// TIA Portal project "PP_0.25AC_new" (V14)

(* hardware
DEVICE "S7-1200 station_1"  S7-1200 Station
   slot 0: "Rack_0"  Rack  V1.0
   slot 1: "PLC_1"  CPU 1215C DC/DC/DC  6ES7 215-1AG40-0XB0  V4.2
   slot 101: "CM 1241 (RS422/485)_1"  6ES7 241-1CH31-0XB0  V1.0
DEVICE "ET 200SP station_1"  ET 200SP-Station
   slot 0: "Rack_0"  Rack  6ES5 710-8MAx1
   slot 0: "IO device_1"  IM 155-6 PN ST  6ES7 155-6AU01-0BN0  V4.1
   slot 1: "AI 8xI 2-,4-wire BA_1"  AI 8xI 2-,4-wire BA  6ES7 134-6GF00-0AA1  V1.0
      slot 1: "AI 8xI 2-,4-wire BA_1"  AI 8xI 2-,4-wire BA
   slot 2: "AI 8xI 2-,4-wire BA_2"  AI 8xI 2-,4-wire BA  6ES7 134-6GF00-0AA1  V1.0
      slot 1: "AI 8xI 2-,4-wire BA_2"  AI 8xI 2-,4-wire BA
   slot 3: "Server module_1"  Server module  6ES7 193-6PA00-0AA0  V1.1
      slot 1: "Server module_1"  Server module
   slot 127: "BA 2xRJ45"  BA 2xRJ45  6ES7 193-6AR00-0AA0  V0.0
      slot 1: "Port_1"  6ES7 193-6AR00-0AA0  V0.0
      slot 2: "Port_2"  6ES7 193-6AR00-0AA0  V0.0
*)

// ===== PLC "PLC_1"  CPU 1215C DC/DC/DC =====

VAR_GLOBAL   // PLC tag table "Default tag table"
   "AI2_0" AT %IW2 : Int;   // Давление нефти на входе, МПа
   "AI2_1" AT %IW4 : Int;   // Давление нефти на выходе, МПа
   "AI2_2" AT %IW6 : Int;   // Давление газа, МПа
   "AI2_3" AT %IW8 : Int;   // Температура на выходе, С
   "AI2_4" AT %IW10 : Int;   // Температура дымовых газов горелки, С
   "AI2_5" AT %IW12 : Int;   // Температура ёмкости, С
   "AI2_6" AT %IW14 : Int;   // Температура в емкости Б1, С ТТ3
   "AI2_7" AT %IW16 : Int;   // Газоанализатор
   "AI3_0" AT %IW18 : Int;   // Резерв
   "AI3_1" AT %IW20 : Int;   // Резерв
   "AI3_2" AT %IW22 : Int;   // Резерв
   "AI3_3" AT %IW24 : Int;   // Резерв
   "AI3_4" AT %IW26 : Int;   // Резерв
   "AI3_5" AT %IW28 : Int;   // Резерв
   "AI3_6" AT %IW30 : Int;   // Резерв
   "AI3_7" AT %IW32 : Int;   // Резерв
   "DI1_0" AT %I0.0 : Bool;   // Сигнализатор уровня MIN ёмкости
   "DI1_1" AT %I0.1 : Bool;   // Сигнализатор уровня MAX ёмкости
   "DI1_2" AT %I0.2 : Bool;   // Клапан 1
   "DI1_3" AT %I0.3 : Bool;   // Клапан 2
   "DI1_4" AT %I0.4 : Bool;   // Резерв
   "DI1_5" AT %I0.5 : Bool;   // Резерв
   "DI1_6" AT %I0.6 : Bool;   // Работа горелки
   "DI1_7" AT %I0.7 : Bool;   // Авария горелки
   "DI1_8" AT %I1.0 : Bool;   // Резерв
   "DI1_9" AT %I1.1 : Bool;   // Резерв
   "DI1_10" AT %I1.2 : Bool;   // Резерв
   "DI1_11" AT %I1.3 : Bool;   // Резерв
   "DI1_12" AT %I1.4 : Bool;   // Резерв
   "DI1_13" AT %I1.5 : Bool;   // Резерв
   "DI2_0" AT %I48.0 : Bool;   // Резерв
   "DI2_1" AT %I48.1 : Bool;   // Резерв
   "DI2_2" AT %I48.2 : Bool;   // Резерв
   "DI2_3" AT %I48.3 : Bool;   // Резерв
   "DI2_4" AT %I48.4 : Bool;   // Резерв
   "DI2_5" AT %I48.5 : Bool;   // Резерв
   "DI2_6" AT %I48.6 : Bool;   // Резерв
   "DI2_7" AT %I48.7 : Bool;   // Резерв
   "DI2_8" AT %I49.0 : Bool;   // Резерв
   "DI2_9" AT %I49.1 : Bool;   // Резерв
   "DI2_10" AT %I49.2 : Bool;   // Резерв
   "DI2_11" AT %I49.3 : Bool;   // Резерв
   "DI2_12" AT %I49.4 : Bool;   // Резерв
   "DI2_13" AT %I49.5 : Bool;   // Резерв
   "DI2_14" AT %I49.6 : Bool;   // Резерв
   "DI2_15" AT %I49.7 : Bool;   // Резерв
   "DO1_0" AT %Q0.0 : Bool;   // ПАСВ оповещатель светозвуковой
   "DO1_1" AT %Q0.1 : Bool;   // ПАСВ оповещатель светозвуковой
   "DO1_2" AT %Q0.2 : Bool;   // Пуск/Стоп горелки
   "DO1_3" AT %Q0.3 : Bool;   // Клапан 1
   "DO1_4" AT %Q0.4 : Bool;   // Клапан 2
   "DO1_5" AT %Q0.5 : Bool;   // ИВНТР
   "DO1_6" AT %Q0.6 : Bool;   // Резерв
   "DO1_7" AT %Q0.7 : Bool;   // Резерв
   "DO1_8" AT %Q1.0 : Bool;   // Резерв
   "DO1_9" AT %Q1.1 : Bool;   // Резерв
   "DO2_0" AT %Q2.0 : Bool;   // Резерв
   "DO2_1" AT %Q2.1 : Bool;   // Резерв
   "DO2_2" AT %Q2.2 : Bool;   // Резерв
   "DO2_3" AT %Q2.3 : Bool;   // Резерв
   "DO2_4" AT %Q2.4 : Bool;   // Резерв
   "DO2_5" AT %Q2.5 : Bool;   // Резерв
   "DO2_6" AT %Q2.6 : Bool;   // Резерв
   "DO2_7" AT %Q2.7 : Bool;   // Резерв
   "DO2_8" AT %Q3.0 : Bool;   // Резерв
   "DO2_9" AT %Q3.1 : Bool;   // Резерв
   "DO2_10" AT %Q3.2 : Bool;   // Резерв
   "DO2_11" AT %Q3.3 : Bool;   // Резерв
   "DO2_12" AT %Q3.4 : Bool;   // Резерв
   "DO2_13" AT %Q3.5 : Bool;   // Резерв
   "DO2_14" AT %Q3.6 : Bool;   // Резерв
   "DO2_15" AT %Q3.7 : Bool;   // Резерв
   "Clock_Byte" AT %MB0 : Byte;
   "Clock_10Hz" AT %M0.0 : Bool;
   "Clock_5Hz" AT %M0.1 : Bool;
   "Clock_2.5Hz" AT %M0.2 : Bool;
   "Clock_2Hz" AT %M0.3 : Bool;
   "Clock_1.25Hz" AT %M0.4 : Bool;
   "Clock_1Hz" AT %M0.5 : Bool;
   "Clock_0.625Hz" AT %M0.6 : Bool;
   "Clock_0.5Hz" AT %M0.7 : Bool;
   "System_Byte" AT %MB1 : Byte;
   "FirstScan" AT %M1.0 : Bool;
   "DiagStatusUpdate" AT %M1.1 : Bool;
   "AlwaysTRUE" AT %M1.2 : Bool;
   "AlwaysFALSE" AT %M1.3 : Bool;
   "EN" AT %M2.0 : Bool;
END_VAR

TYPE "Burner_DT"
VERSION : 0.1
   STRUCT
      State : Int;
      CMD_in : Int;
      Alarm : Int;
   END_STRUCT;
END_TYPE

TYPE "AI_DT"
VERSION : 0.1
   STRUCT
      Hihi_Value : Real;   // Уставка: Hihi
      High_Value : Real;   // Уставка: High
      Low_Value : Real;   // Уставка: Low
      Lolo_Value : Real;   // Уставка: Lolo
      MIN_Current : Real;   // Настройка: Минимальное входное значение тока
      MAX_Current : Real;   // Настройка: Максимальное входное значение тока
      MAX_Value : Real;   // Настройка: Максимальное значение измеряемой величины
      MIN_Value : Real;   // Настройка: Минимальное значение измеряемой величины
      Underflow_RAW : Real;   // Настройка: Значение кода ацп при обрыве
      Overflow_RAW : Real;   // Настройка: Значение кода ацп при зашкале
      SCALED : Real;   // Выход: Масштабированное в инженерные единицы значение входного сигнала
      ING_Value : Real;   // Выход: Токовое значение датчика
      Manual_Value : Real;   // Значение, введенное вручную
      Alarm_Delay : Int;   // Настройка: Задержка срабатывания аварий
      Warning_Delay : Int;   // Настройка: Задержка срабатывания предупреждений
      AVG_Delay : Real;   // Настройка: Зона нечувствительности
      Underflow_Delay : Int;   // Настройка: Задержка отображения обрыва датчика
      Overflow_Delay : Int;   // Настройка: Задержка отображения неисправности датчика
      State : Word;   // Выход: Состояние датчика
      Modeee : Word;   // Настройка: Режим работы датчика
      bools : Word;   // Все булевы параметры AI
      AI_RAW_MIN : Int;   // Мин кода ацп
      AI_RAW_MAX : Int;   // Макс кода ацп
      Hihi_EN : Bool;   // Разрешение на сработку
      High_EN : Bool;   // Разрешение на сработку
      Low_En : Bool;   // Разрешение на сработку
      Lolo_EN : Bool;   // Разрешение на сработку
   END_STRUCT;
END_TYPE

TYPE "Ustavki"
   STRUCT
      Hihi : Bool;
      Hi : Bool;
      Lo : Bool;
      Lolo : Bool;
   END_STRUCT;
END_TYPE

TYPE "PAZ_DT"
VERSION : 0.1
   STRUCT
      Alarm_EN : Bool;
      ZP_EN : Bool;
      IN : Bool;
      Alarm_out : Bool;
      ZP_out : Bool;
   END_STRUCT;
END_TYPE

TYPE "Hiter"
VERSION : 0.1
   STRUCT
      Mode : Bool;
      T_state : Int;
      CMD : Bool;
      Avar_stop : Bool;
   END_STRUCT;
END_TYPE

TYPE "DI_DT"
VERSION : 0.1
   STRUCT
      Time_ON : Int;   // Время перехода OFF->ON
      Time_OFF : Int;   // Время перехода ON->OFF
      Input : Bool;   // Значение с модуля
      Disable : Bool;   // Запрет обработки канала
      Invert : Bool;   // Инертирование канала
      Output : Bool;   // Значение канала для логики
   END_STRUCT;
END_TYPE

TYPE "Valve_DT"
VERSION : 0.1
   STRUCT
      State : Int;
      State_ctrl : Bool;
      Alarm : Int;
      Cmd_in : Int;
      Cmd_out : Bool;
      bools : Int;
      Deblock : Bool;
   END_STRUCT;
END_TYPE

TYPE "Valve_ctrl_DT"
VERSION : 0.1
   STRUCT
      State : Int;
      Cmd_in : Int;
      TIME_shod : Int;
      TIME_hod : Int;
      bools : DWord;
   END_STRUCT;
END_TYPE

TYPE "DO_DT"
VERSION : 0.1
   STRUCT
      Time_ON : Int;   // Время перехода OFF->ON
      Time_OFF : Int;   // Время перехода ON->OFF
      Input : Bool;   // Значение от логики
      Disable : Bool;   // Запрет обработки канала
      Invert : Bool;   // Инертирование канала
      Output : Bool;   // Значение на модуль
   END_STRUCT;
END_TYPE

DATA_BLOCK "PLC_Signals_DB"   // DB1
{ S7_Optimized_Access := 'FALSE' }
VERSION : 0.1
   VAR
      AI_2_0 : Struct   // Давление на выходе
         Hihi_Value : Real := 70.0;   // Уставка: Hihi
         High_Value : Real := 60.0;   // Уставка: High
         Low_Value : Real := 30.0;   // Уставка: Low
         Lolo_Value : Real := 20.0;   // Уставка: Lolo
         MIN_Current : Real := 4.0;   // Настройка: Минимальное входное значение тока
         MAX_Current : Real := 20.0;   // Настройка: Максимальное входное значение тока
         MAX_Value : Real := 1.0;   // Настройка: Максимальное значение измеряемой величины
         MIN_Value : Real := 0.0;   // Настройка: Минимальное значение измеряемой величины
         Underflow_RAW : Real := -10.0;   // Настройка: Значение кода ацп при обрыве
         Overflow_RAW : Real := 27650.0;   // Настройка: Значение кода ацп при зашкале
         SCALED : Real := 0.0;   // Выход: Масштабированное в инженерные единицы значение входного сигнала
         ING_Value : Real := 0.0;   // Выход: Токовое значение датчика
         Manual_Value : Real := 50.0;   // Значение, введенное вручную
         Alarm_Delay : Int := 0;   // Настройка: Задержка срабатывания аварий
         Warning_Delay : Int := 0;   // Настройка: Задержка срабатывания предупреждений
         AVG_Delay : Real := 0.0;   // Настройка: Зона нечувствительности
         Underflow_Delay : Int := 0;   // Настройка: Задержка отображения обрыва датчика
         Overflow_Delay : Int := 0;   // Настройка: Задержка отображения неисправности датчика
         StateHMI : Int;
         State : Word := 16#0;   // Выход: Состояние датчика
         Modeee : Word := 16#1;   // Настройка: Режим работы датчика
         bools : Word := 16#0;   // Все булевы параметры AI
         AI_RAW_MIN : Int := 0;   // Мин кода ацп
         AI_RAW_MAX : Int := 27648;   // Макс кода ацп
         Hihi_EN : Bool := false;   // Разрешение на сработку
         High_EN : Bool := false;   // Разрешение на сработку
         Low_En : Bool := false;   // Разрешение на сработку
         Lolo_EN : Bool := false;   // Разрешение на сработку
      END_STRUCT;
      AI_2_1 : Struct   // Давление на входе
         Hihi_Value : Real := 70.0;   // Уставка: Hihi
         High_Value : Real := 60.0;   // Уставка: High
         Low_Value : Real := 30.0;   // Уставка: Low
         Lolo_Value : Real := 20.0;   // Уставка: Lolo
         MIN_Current : Real := 4.0;   // Настройка: Минимальное входное значение тока
         MAX_Current : Real := 20.0;   // Настройка: Максимальное входное значение тока
         MAX_Value : Real := 1.0;   // Настройка: Максимальное значение измеряемой величины
         MIN_Value : Real := 0.0;   // Настройка: Минимальное значение измеряемой величины
         Underflow_RAW : Real := -10.0;   // Настройка: Значение кода ацп при обрыве
         Overflow_RAW : Real := 27650.0;   // Настройка: Значение кода ацп при зашкале
         SCALED : Real := 0.0;   // Выход: Масштабированное в инженерные единицы значение входного сигнала
         ING_Value : Real := 0.0;   // Выход: Токовое значение датчика
         Manual_Value : Real := 50.0;   // Значение, введенное вручную
         Alarm_Delay : Int := 0;   // Настройка: Задержка срабатывания аварий
         Warning_Delay : Int := 0;   // Настройка: Задержка срабатывания предупреждений
         AVG_Delay : Real := 0.0;   // Настройка: Зона нечувствительности
         Underflow_Delay : Int := 0;   // Настройка: Задержка отображения обрыва датчика
         Overflow_Delay : Int := 0;   // Настройка: Задержка отображения неисправности датчика
         StateHMI : Int;
         State : Word := 16#0;   // Выход: Состояние датчика
         Modeee : Word := 16#1;   // Настройка: Режим работы датчика
         bools : Word := 16#0;   // Все булевы параметры AI
         AI_RAW_MIN : Int := 0;   // Мин кода ацп
         AI_RAW_MAX : Int := 27648;   // Макс кода ацп
         Hihi_EN : Bool := false;   // Разрешение на сработку
         High_EN : Bool := false;   // Разрешение на сработку
         Low_En : Bool := false;   // Разрешение на сработку
         Lolo_EN : Bool := false;   // Разрешение на сработку
      END_STRUCT;
      AI_2_2 : Struct   // Датчик давления газа
         Hihi_Value : Real := 70.0;   // Уставка: Hihi
         High_Value : Real := 60.0;   // Уставка: High
         Low_Value : Real := 30.0;   // Уставка: Low
         Lolo_Value : Real := 20.0;   // Уставка: Lolo
         MIN_Current : Real := 4.0;   // Настройка: Минимальное входное значение тока
         MAX_Current : Real := 20.0;   // Настройка: Максимальное входное значение тока
         MAX_Value : Real := 1.0;   // Настройка: Максимальное значение измеряемой величины
         MIN_Value : Real := 0.0;   // Настройка: Минимальное значение измеряемой величины
         Underflow_RAW : Real := -10.0;   // Настройка: Значение кода ацп при обрыве
         Overflow_RAW : Real := 27650.0;   // Настройка: Значение кода ацп при зашкале
         SCALED : Real := 0.0;   // Выход: Масштабированное в инженерные единицы значение входного сигнала
         ING_Value : Real := 0.0;   // Выход: Токовое значение датчика
         Manual_Value : Real := 50.0;   // Значение, введенное вручную
         Alarm_Delay : Int := 0;   // Настройка: Задержка срабатывания аварий
         Warning_Delay : Int := 0;   // Настройка: Задержка срабатывания предупреждений
         AVG_Delay : Real := 0.0;   // Настройка: Зона нечувствительности
         Underflow_Delay : Int := 0;   // Настройка: Задержка отображения обрыва датчика
         Overflow_Delay : Int := 0;   // Настройка: Задержка отображения неисправности датчика
         StateHMI : Int;
         State : Word := 16#0;   // Выход: Состояние датчика
         Modeee : Word := 16#1;   // Настройка: Режим работы датчика
         bools : Word := 16#0;   // Все булевы параметры AI
         AI_RAW_MIN : Int := 0;   // Мин кода ацп
         AI_RAW_MAX : Int := 27648;   // Макс кода ацп
         Hihi_EN : Bool := false;   // Разрешение на сработку
         High_EN : Bool := false;   // Разрешение на сработку
         Low_En : Bool := false;   // Разрешение на сработку
         Lolo_EN : Bool := false;   // Разрешение на сработку
      END_STRUCT;
      AI_2_3 : Struct   // Температура на выходе
         Hihi_Value : Real := 70.0;   // Уставка: Hihi
         High_Value : Real := 60.0;   // Уставка: High
         Low_Value : Real := 30.0;   // Уставка: Low
         Lolo_Value : Real := 20.0;   // Уставка: Lolo
         MIN_Current : Real := 4.0;   // Настройка: Минимальное входное значение тока
         MAX_Current : Real := 20.0;   // Настройка: Максимальное входное значение тока
         MAX_Value : Real := 100.0;   // Настройка: Максимальное значение измеряемой величины
         MIN_Value : Real := -50.0;   // Настройка: Минимальное значение измеряемой величины
         Underflow_RAW : Real := -10.0;   // Настройка: Значение кода ацп при обрыве
         Overflow_RAW : Real := 27650.0;   // Настройка: Значение кода ацп при зашкале
         SCALED : Real := 0.0;   // Выход: Масштабированное в инженерные единицы значение входного сигнала
         ING_Value : Real := 0.0;   // Выход: Токовое значение датчика
         Manual_Value : Real := 50.0;   // Значение, введенное вручную
         Alarm_Delay : Int := 0;   // Настройка: Задержка срабатывания аварий
         Warning_Delay : Int := 0;   // Настройка: Задержка срабатывания предупреждений
         AVG_Delay : Real := 0.0;   // Настройка: Зона нечувствительности
         Underflow_Delay : Int := 0;   // Настройка: Задержка отображения обрыва датчика
         Overflow_Delay : Int := 0;   // Настройка: Задержка отображения неисправности датчика
         StateHMI : Int;
         State : Word := 16#0;   // Выход: Состояние датчика
         Modeee : Word := 16#1;   // Настройка: Режим работы датчика
         bools : Word := 16#0;   // Все булевы параметры AI
         AI_RAW_MIN : Int := 0;   // Мин кода ацп
         AI_RAW_MAX : Int := 27648;   // Макс кода ацп
         Hihi_EN : Bool := false;   // Разрешение на сработку
         High_EN : Bool := false;   // Разрешение на сработку
         Low_En : Bool := false;   // Разрешение на сработку
         Lolo_EN : Bool := false;   // Разрешение на сработку
      END_STRUCT;
      AI_2_4 : Struct   // Температура дымовых газов
         Hihi_Value : Real := 70.0;   // Уставка: Hihi
         High_Value : Real := 60.0;   // Уставка: High
         Low_Value : Real := 30.0;   // Уставка: Low
         Lolo_Value : Real := 20.0;   // Уставка: Lolo
         MIN_Current : Real := 4.0;   // Настройка: Минимальное входное значение тока
         MAX_Current : Real := 20.0;   // Настройка: Максимальное входное значение тока
         MAX_Value : Real := 500.0;   // Настройка: Максимальное значение измеряемой величины
         MIN_Value : Real := -50.0;   // Настройка: Минимальное значение измеряемой величины
         Underflow_RAW : Real := -10.0;   // Настройка: Значение кода ацп при обрыве
         Overflow_RAW : Real := 27650.0;   // Настройка: Значение кода ацп при зашкале
         SCALED : Real := 0.0;   // Выход: Масштабированное в инженерные единицы значение входного сигнала
         ING_Value : Real := 0.0;   // Выход: Токовое значение датчика
         Manual_Value : Real := 50.0;   // Значение, введенное вручную
         Alarm_Delay : Int := 0;   // Настройка: Задержка срабатывания аварий
         Warning_Delay : Int := 0;   // Настройка: Задержка срабатывания предупреждений
         AVG_Delay : Real := 0.0;   // Настройка: Зона нечувствительности
         Underflow_Delay : Int := 0;   // Настройка: Задержка отображения обрыва датчика
         Overflow_Delay : Int := 0;   // Настройка: Задержка отображения неисправности датчика
         StateHMI : Int;
         State : Word := 16#0;   // Выход: Состояние датчика
         Modeee : Word := 16#1;   // Настройка: Режим работы датчика
         bools : Word := 16#0;   // Все булевы параметры AI
         AI_RAW_MIN : Int := 0;   // Мин кода ацп
         AI_RAW_MAX : Int := 27648;   // Макс кода ацп
         Hihi_EN : Bool := false;   // Разрешение на сработку
         High_EN : Bool := false;   // Разрешение на сработку
         Low_En : Bool := false;   // Разрешение на сработку
         Lolo_EN : Bool := false;   // Разрешение на сработку
      END_STRUCT;
      AI_2_5 : Struct   // Температура ёмкости
         Hihi_Value : Real := 70.0;   // Уставка: Hihi
         High_Value : Real := 60.0;   // Уставка: High
         Low_Value : Real := 30.0;   // Уставка: Low
         Lolo_Value : Real := 20.0;   // Уставка: Lolo
         MIN_Current : Real := 4.0;   // Настройка: Минимальное входное значение тока
         MAX_Current : Real := 20.0;   // Настройка: Максимальное входное значение тока
         MAX_Value : Real := 100.0;   // Настройка: Максимальное значение измеряемой величины
         MIN_Value : Real := -50.0;   // Настройка: Минимальное значение измеряемой величины
         Underflow_RAW : Real := -10.0;   // Настройка: Значение кода ацп при обрыве
         Overflow_RAW : Real := 27650.0;   // Настройка: Значение кода ацп при зашкале
         SCALED : Real := 0.0;   // Выход: Масштабированное в инженерные единицы значение входного сигнала
         ING_Value : Real := 0.0;   // Выход: Токовое значение датчика
         Manual_Value : Real := 50.0;   // Значение, введенное вручную
         Alarm_Delay : Int := 0;   // Настройка: Задержка срабатывания аварий
         Warning_Delay : Int := 0;   // Настройка: Задержка срабатывания предупреждений
         AVG_Delay : Real := 0.0;   // Настройка: Зона нечувствительности
         Underflow_Delay : Int := 0;   // Настройка: Задержка отображения обрыва датчика
         Overflow_Delay : Int := 0;   // Настройка: Задержка отображения неисправности датчика
         StateHMI : Int;
         State : Word := 16#0;   // Выход: Состояние датчика
         Modeee : Word := 16#1;   // Настройка: Режим работы датчика
         bools : Word := 16#0;   // Все булевы параметры AI
         AI_RAW_MIN : Int := 0;   // Мин кода ацп
         AI_RAW_MAX : Int := 27648;   // Макс кода ацп
         Hihi_EN : Bool := false;   // Разрешение на сработку
         High_EN : Bool := false;   // Разрешение на сработку
         Low_En : Bool := false;   // Разрешение на сработку
         Lolo_EN : Bool := false;   // Разрешение на сработку
      END_STRUCT;
      AI_2_6 : Struct   // Газоанализатор ДГС
         Hihi_Value : Real := 70.0;   // Уставка: Hihi
         High_Value : Real := 60.0;   // Уставка: High
         Low_Value : Real := 30.0;   // Уставка: Low
         Lolo_Value : Real := 20.0;   // Уставка: Lolo
         MIN_Current : Real := 4.0;   // Настройка: Минимальное входное значение тока
         MAX_Current : Real := 20.0;   // Настройка: Максимальное входное значение тока
         MAX_Value : Real := 100.0;   // Настройка: Максимальное значение измеряемой величины
         MIN_Value : Real := -50.0;   // Настройка: Минимальное значение измеряемой величины
         Underflow_RAW : Real := -10.0;   // Настройка: Значение кода ацп при обрыве
         Overflow_RAW : Real := 27650.0;   // Настройка: Значение кода ацп при зашкале
         SCALED : Real := 0.0;   // Выход: Масштабированное в инженерные единицы значение входного сигнала
         ING_Value : Real := 0.0;   // Выход: Токовое значение датчика
         Manual_Value : Real := 50.0;   // Значение, введенное вручную
         Alarm_Delay : Int := 0;   // Настройка: Задержка срабатывания аварий
         Warning_Delay : Int := 0;   // Настройка: Задержка срабатывания предупреждений
         AVG_Delay : Real := 0.0;   // Настройка: Зона нечувствительности
         Underflow_Delay : Int := 0;   // Настройка: Задержка отображения обрыва датчика
         Overflow_Delay : Int := 0;   // Настройка: Задержка отображения неисправности датчика
         StateHMI : Int;
         State : Word := 16#0;   // Выход: Состояние датчика
         Modeee : Word := 16#1;   // Настройка: Режим работы датчика
         bools : Word := 16#0;   // Все булевы параметры AI
         AI_RAW_MIN : Int := 0;   // Мин кода ацп
         AI_RAW_MAX : Int := 27648;   // Макс кода ацп
         Hihi_EN : Bool := false;   // Разрешение на сработку
         High_EN : Bool := false;   // Разрешение на сработку
         Low_En : Bool := false;   // Разрешение на сработку
         Lolo_EN : Bool := false;   // Разрешение на сработку
      END_STRUCT;
      AI_2_7 : Struct   // Резерв
         Hihi_Value : Real := 70.0;   // Уставка: Hihi
         High_Value : Real := 60.0;   // Уставка: High
         Low_Value : Real := 30.0;   // Уставка: Low
         Lolo_Value : Real := 20.0;   // Уставка: Lolo
         MIN_Current : Real := 4.0;   // Настройка: Минимальное входное значение тока
         MAX_Current : Real := 20.0;   // Настройка: Максимальное входное значение тока
         MAX_Value : Real := 100.0;   // Настройка: Максимальное значение измеряемой величины
         MIN_Value : Real := 0.0;   // Настройка: Минимальное значение измеряемой величины
         Underflow_RAW : Real := -10.0;   // Настройка: Значение кода ацп при обрыве
         Overflow_RAW : Real := 27650.0;   // Настройка: Значение кода ацп при зашкале
         SCALED : Real := 0.0;   // Выход: Масштабированное в инженерные единицы значение входного сигнала
         ING_Value : Real := 0.0;   // Выход: Токовое значение датчика
         Manual_Value : Real := 50.0;   // Значение, введенное вручную
         Alarm_Delay : Int := 0;   // Настройка: Задержка срабатывания аварий
         Warning_Delay : Int := 0;   // Настройка: Задержка срабатывания предупреждений
         AVG_Delay : Real := 0.0;   // Настройка: Зона нечувствительности
         Underflow_Delay : Int := 0;   // Настройка: Задержка отображения обрыва датчика
         Overflow_Delay : Int := 0;   // Настройка: Задержка отображения неисправности датчика
         StateHMI : Int;
         State : Word := 16#0;   // Выход: Состояние датчика
         Modeee : Word := 16#1;   // Настройка: Режим работы датчика
         bools : Word := 16#0;   // Все булевы параметры AI
         AI_RAW_MIN : Int := 0;   // Мин кода ацп
         AI_RAW_MAX : Int := 27648;   // Макс кода ацп
         Hihi_EN : Bool := false;   // Разрешение на сработку
         High_EN : Bool := false;   // Разрешение на сработку
         Low_En : Bool := false;   // Разрешение на сработку
         Lolo_EN : Bool := false;   // Разрешение на сработку
      END_STRUCT;
      AI_3_0 : Struct   // Резерв
         Hihi_Value : Real := 70.0;   // Уставка: Hihi
         High_Value : Real := 60.0;   // Уставка: High
         Low_Value : Real := 30.0;   // Уставка: Low
         Lolo_Value : Real := 20.0;   // Уставка: Lolo
         MIN_Current : Real := 4.0;   // Настройка: Минимальное входное значение тока
         MAX_Current : Real := 20.0;   // Настройка: Максимальное входное значение тока
         MAX_Value : Real := 100.0;   // Настройка: Максимальное значение измеряемой величины
         MIN_Value : Real := 0.0;   // Настройка: Минимальное значение измеряемой величины
         Underflow_RAW : Real := -10.0;   // Настройка: Значение кода ацп при обрыве
         Overflow_RAW : Real := 27650.0;   // Настройка: Значение кода ацп при зашкале
         SCALED : Real := 0.0;   // Выход: Масштабированное в инженерные единицы значение входного сигнала
         ING_Value : Real := 0.0;   // Выход: Токовое значение датчика
         Manual_Value : Real := 50.0;   // Значение, введенное вручную
         Alarm_Delay : Int := 0;   // Настройка: Задержка срабатывания аварий
         Warning_Delay : Int := 0;   // Настройка: Задержка срабатывания предупреждений
         AVG_Delay : Real := 0.0;   // Настройка: Зона нечувствительности
         Underflow_Delay : Int := 0;   // Настройка: Задержка отображения обрыва датчика
         Overflow_Delay : Int := 0;   // Настройка: Задержка отображения неисправности датчика
         StateHMI : Int;
         State : Word := 16#0;   // Выход: Состояние датчика
         Modeee : Word := 16#1;   // Настройка: Режим работы датчика
         bools : Word := 16#0;   // Все булевы параметры AI
         AI_RAW_MIN : Int := 0;   // Мин кода ацп
         AI_RAW_MAX : Int := 27648;   // Макс кода ацп
         Hihi_EN : Bool := false;   // Разрешение на сработку
         High_EN : Bool := false;   // Разрешение на сработку
         Low_En : Bool := false;   // Разрешение на сработку
         Lolo_EN : Bool := false;   // Разрешение на сработку
      END_STRUCT;
      AI_3_1 : Struct   // Резерв
         Hihi_Value : Real := 70.0;   // Уставка: Hihi
         High_Value : Real := 60.0;   // Уставка: High
         Low_Value : Real := 30.0;   // Уставка: Low
         Lolo_Value : Real := 20.0;   // Уставка: Lolo
         MIN_Current : Real := 4.0;   // Настройка: Минимальное входное значение тока
         MAX_Current : Real := 20.0;   // Настройка: Максимальное входное значение тока
         MAX_Value : Real := 100.0;   // Настройка: Максимальное значение измеряемой величины
         MIN_Value : Real := 0.0;   // Настройка: Минимальное значение измеряемой величины
         Underflow_RAW : Real := -10.0;   // Настройка: Значение кода ацп при обрыве
         Overflow_RAW : Real := 27650.0;   // Настройка: Значение кода ацп при зашкале
         SCALED : Real := 0.0;   // Выход: Масштабированное в инженерные единицы значение входного сигнала
         ING_Value : Real := 0.0;   // Выход: Токовое значение датчика
         Manual_Value : Real := 50.0;   // Значение, введенное вручную
         Alarm_Delay : Int := 0;   // Настройка: Задержка срабатывания аварий
         Warning_Delay : Int := 0;   // Настройка: Задержка срабатывания предупреждений
         AVG_Delay : Real := 0.0;   // Настройка: Зона нечувствительности
         Underflow_Delay : Int := 0;   // Настройка: Задержка отображения обрыва датчика
         Overflow_Delay : Int := 0;   // Настройка: Задержка отображения неисправности датчика
         StateHMI : Int;
         State : Word := 16#0;   // Выход: Состояние датчика
         Modeee : Word := 16#1;   // Настройка: Режим работы датчика
         bools : Word := 16#0;   // Все булевы параметры AI
         AI_RAW_MIN : Int := 0;   // Мин кода ацп
         AI_RAW_MAX : Int := 27648;   // Макс кода ацп
         Hihi_EN : Bool := false;   // Разрешение на сработку
         High_EN : Bool := false;   // Разрешение на сработку
         Low_En : Bool := false;   // Разрешение на сработку
         Lolo_EN : Bool := false;   // Разрешение на сработку
      END_STRUCT;
      AI_3_2 : Struct   // Резерв
         Hihi_Value : Real := 70.0;   // Уставка: Hihi
         High_Value : Real := 60.0;   // Уставка: High
         Low_Value : Real := 30.0;   // Уставка: Low
         Lolo_Value : Real := 20.0;   // Уставка: Lolo
         MIN_Current : Real := 4.0;   // Настройка: Минимальное входное значение тока
         MAX_Current : Real := 20.0;   // Настройка: Максимальное входное значение тока
         MAX_Value : Real := 100.0;   // Настройка: Максимальное значение измеряемой величины
         MIN_Value : Real := 0.0;   // Настройка: Минимальное значение измеряемой величины
         Underflow_RAW : Real := -10.0;   // Настройка: Значение кода ацп при обрыве
         Overflow_RAW : Real := 27650.0;   // Настройка: Значение кода ацп при зашкале
         SCALED : Real := 0.0;   // Выход: Масштабированное в инженерные единицы значение входного сигнала
         ING_Value : Real := 0.0;   // Выход: Токовое значение датчика
         Manual_Value : Real := 50.0;   // Значение, введенное вручную
         Alarm_Delay : Int := 0;   // Настройка: Задержка срабатывания аварий
         Warning_Delay : Int := 0;   // Настройка: Задержка срабатывания предупреждений
         AVG_Delay : Real := 0.0;   // Настройка: Зона нечувствительности
         Underflow_Delay : Int := 0;   // Настройка: Задержка отображения обрыва датчика
         Overflow_Delay : Int := 0;   // Настройка: Задержка отображения неисправности датчика
         StateHMI : Int;
         State : Word := 16#0;   // Выход: Состояние датчика
         Modeee : Word := 16#1;   // Настройка: Режим работы датчика
         bools : Word := 16#0;   // Все булевы параметры AI
         AI_RAW_MIN : Int := 0;   // Мин кода ацп
         AI_RAW_MAX : Int := 27648;   // Макс кода ацп
         Hihi_EN : Bool := false;   // Разрешение на сработку
         High_EN : Bool := false;   // Разрешение на сработку
         Low_En : Bool := false;   // Разрешение на сработку
         Lolo_EN : Bool := false;   // Разрешение на сработку
      END_STRUCT;
      AI_3_3 : Struct   // Резерв
         Hihi_Value : Real := 70.0;   // Уставка: Hihi
         High_Value : Real := 60.0;   // Уставка: High
         Low_Value : Real := 30.0;   // Уставка: Low
         Lolo_Value : Real := 20.0;   // Уставка: Lolo
         MIN_Current : Real := 4.0;   // Настройка: Минимальное входное значение тока
         MAX_Current : Real := 20.0;   // Настройка: Максимальное входное значение тока
         MAX_Value : Real := 100.0;   // Настройка: Максимальное значение измеряемой величины
         MIN_Value : Real := 0.0;   // Настройка: Минимальное значение измеряемой величины
         Underflow_RAW : Real := -10.0;   // Настройка: Значение кода ацп при обрыве
         Overflow_RAW : Real := 27650.0;   // Настройка: Значение кода ацп при зашкале
         SCALED : Real := 0.0;   // Выход: Масштабированное в инженерные единицы значение входного сигнала
         ING_Value : Real := 0.0;   // Выход: Токовое значение датчика
         Manual_Value : Real := 50.0;   // Значение, введенное вручную
         Alarm_Delay : Int := 0;   // Настройка: Задержка срабатывания аварий
         Warning_Delay : Int := 0;   // Настройка: Задержка срабатывания предупреждений
         AVG_Delay : Real := 0.0;   // Настройка: Зона нечувствительности
         Underflow_Delay : Int := 0;   // Настройка: Задержка отображения обрыва датчика
         Overflow_Delay : Int := 0;   // Настройка: Задержка отображения неисправности датчика
         StateHMI : Int;
         State : Word := 16#0;   // Выход: Состояние датчика
         Modeee : Word := 16#1;   // Настройка: Режим работы датчика
         bools : Word := 16#0;   // Все булевы параметры AI
         AI_RAW_MIN : Int := 0;   // Мин кода ацп
         AI_RAW_MAX : Int := 27648;   // Макс кода ацп
         Hihi_EN : Bool := false;   // Разрешение на сработку
         High_EN : Bool := false;   // Разрешение на сработку
         Low_En : Bool := false;   // Разрешение на сработку
         Lolo_EN : Bool := false;   // Разрешение на сработку
      END_STRUCT;
      AI_3_4 : Struct   // Резерв
         Hihi_Value : Real := 70.0;   // Уставка: Hihi
         High_Value : Real := 60.0;   // Уставка: High
         Low_Value : Real := 30.0;   // Уставка: Low
         Lolo_Value : Real := 20.0;   // Уставка: Lolo
         MIN_Current : Real := 4.0;   // Настройка: Минимальное входное значение тока
         MAX_Current : Real := 20.0;   // Настройка: Максимальное входное значение тока
         MAX_Value : Real := 100.0;   // Настройка: Максимальное значение измеряемой величины
         MIN_Value : Real := 0.0;   // Настройка: Минимальное значение измеряемой величины
         Underflow_RAW : Real := -10.0;   // Настройка: Значение кода ацп при обрыве
         Overflow_RAW : Real := 27650.0;   // Настройка: Значение кода ацп при зашкале
         SCALED : Real := 0.0;   // Выход: Масштабированное в инженерные единицы значение входного сигнала
         ING_Value : Real := 0.0;   // Выход: Токовое значение датчика
         Manual_Value : Real := 50.0;   // Значение, введенное вручную
         Alarm_Delay : Int := 0;   // Настройка: Задержка срабатывания аварий
         Warning_Delay : Int := 0;   // Настройка: Задержка срабатывания предупреждений
         AVG_Delay : Real := 0.0;   // Настройка: Зона нечувствительности
         Underflow_Delay : Int := 0;   // Настройка: Задержка отображения обрыва датчика
         Overflow_Delay : Int := 0;   // Настройка: Задержка отображения неисправности датчика
         StateHMI : Int;
         State : Word := 16#0;   // Выход: Состояние датчика
         Modeee : Word := 16#1;   // Настройка: Режим работы датчика
         bools : Word := 16#0;   // Все булевы параметры AI
         AI_RAW_MIN : Int := 0;   // Мин кода ацп
         AI_RAW_MAX : Int := 27648;   // Макс кода ацп
         Hihi_EN : Bool := false;   // Разрешение на сработку
         High_EN : Bool := false;   // Разрешение на сработку
         Low_En : Bool := false;   // Разрешение на сработку
         Lolo_EN : Bool := false;   // Разрешение на сработку
      END_STRUCT;
      AI_3_5 : Struct   // Резерв
         Hihi_Value : Real := 70.0;   // Уставка: Hihi
         High_Value : Real := 60.0;   // Уставка: High
         Low_Value : Real := 30.0;   // Уставка: Low
         Lolo_Value : Real := 20.0;   // Уставка: Lolo
         MIN_Current : Real := 4.0;   // Настройка: Минимальное входное значение тока
         MAX_Current : Real := 20.0;   // Настройка: Максимальное входное значение тока
         MAX_Value : Real := 100.0;   // Настройка: Максимальное значение измеряемой величины
         MIN_Value : Real := 0.0;   // Настройка: Минимальное значение измеряемой величины
         Underflow_RAW : Real := -10.0;   // Настройка: Значение кода ацп при обрыве
         Overflow_RAW : Real := 27650.0;   // Настройка: Значение кода ацп при зашкале
         SCALED : Real := 0.0;   // Выход: Масштабированное в инженерные единицы значение входного сигнала
         ING_Value : Real := 0.0;   // Выход: Токовое значение датчика
         Manual_Value : Real := 50.0;   // Значение, введенное вручную
         Alarm_Delay : Int := 0;   // Настройка: Задержка срабатывания аварий
         Warning_Delay : Int := 0;   // Настройка: Задержка срабатывания предупреждений
         AVG_Delay : Real := 0.0;   // Настройка: Зона нечувствительности
         Underflow_Delay : Int := 0;   // Настройка: Задержка отображения обрыва датчика
         Overflow_Delay : Int := 0;   // Настройка: Задержка отображения неисправности датчика
         StateHMI : Int;
         State : Word := 16#0;   // Выход: Состояние датчика
         Modeee : Word := 16#1;   // Настройка: Режим работы датчика
         bools : Word := 16#0;   // Все булевы параметры AI
         AI_RAW_MIN : Int := 0;   // Мин кода ацп
         AI_RAW_MAX : Int := 27648;   // Макс кода ацп
         Hihi_EN : Bool := false;   // Разрешение на сработку
         High_EN : Bool := false;   // Разрешение на сработку
         Low_En : Bool := false;   // Разрешение на сработку
         Lolo_EN : Bool := false;   // Разрешение на сработку
      END_STRUCT;
      AI_3_6 : Struct   // Резерв
         Hihi_Value : Real := 70.0;   // Уставка: Hihi
         High_Value : Real := 60.0;   // Уставка: High
         Low_Value : Real := 30.0;   // Уставка: Low
         Lolo_Value : Real := 20.0;   // Уставка: Lolo
         MIN_Current : Real := 4.0;   // Настройка: Минимальное входное значение тока
         MAX_Current : Real := 20.0;   // Настройка: Максимальное входное значение тока
         MAX_Value : Real := 100.0;   // Настройка: Максимальное значение измеряемой величины
         MIN_Value : Real := 0.0;   // Настройка: Минимальное значение измеряемой величины
         Underflow_RAW : Real := -10.0;   // Настройка: Значение кода ацп при обрыве
         Overflow_RAW : Real := 27650.0;   // Настройка: Значение кода ацп при зашкале
         SCALED : Real := 0.0;   // Выход: Масштабированное в инженерные единицы значение входного сигнала
         ING_Value : Real := 0.0;   // Выход: Токовое значение датчика
         Manual_Value : Real := 50.0;   // Значение, введенное вручную
         Alarm_Delay : Int := 0;   // Настройка: Задержка срабатывания аварий
         Warning_Delay : Int := 0;   // Настройка: Задержка срабатывания предупреждений
         AVG_Delay : Real := 0.0;   // Настройка: Зона нечувствительности
         Underflow_Delay : Int := 0;   // Настройка: Задержка отображения обрыва датчика
         Overflow_Delay : Int := 0;   // Настройка: Задержка отображения неисправности датчика
         StateHMI : Int;
         State : Word := 16#0;   // Выход: Состояние датчика
         Modeee : Word := 16#1;   // Настройка: Режим работы датчика
         bools : Word := 16#0;   // Все булевы параметры AI
         AI_RAW_MIN : Int := 0;   // Мин кода ацп
         AI_RAW_MAX : Int := 27648;   // Макс кода ацп
         Hihi_EN : Bool := false;   // Разрешение на сработку
         High_EN : Bool := false;   // Разрешение на сработку
         Low_En : Bool := false;   // Разрешение на сработку
         Lolo_EN : Bool := false;   // Разрешение на сработку
      END_STRUCT;
      AI_3_7 : Struct   // Резерв
         Hihi_Value : Real := 70.0;   // Уставка: Hihi
         High_Value : Real := 60.0;   // Уставка: High
         Low_Value : Real := 30.0;   // Уставка: Low
         Lolo_Value : Real := 20.0;   // Уставка: Lolo
         MIN_Current : Real := 4.0;   // Настройка: Минимальное входное значение тока
         MAX_Current : Real := 20.0;   // Настройка: Максимальное входное значение тока
         MAX_Value : Real := 100.0;   // Настройка: Максимальное значение измеряемой величины
         MIN_Value : Real := 0.0;   // Настройка: Минимальное значение измеряемой величины
         Underflow_RAW : Real := -10.0;   // Настройка: Значение кода ацп при обрыве
         Overflow_RAW : Real := 27650.0;   // Настройка: Значение кода ацп при зашкале
         SCALED : Real := 0.0;   // Выход: Масштабированное в инженерные единицы значение входного сигнала
         ING_Value : Real := 0.0;   // Выход: Токовое значение датчика
         Manual_Value : Real := 50.0;   // Значение, введенное вручную
         Alarm_Delay : Int := 0;   // Настройка: Задержка срабатывания аварий
         Warning_Delay : Int := 0;   // Настройка: Задержка срабатывания предупреждений
         AVG_Delay : Real := 0.0;   // Настройка: Зона нечувствительности
         Underflow_Delay : Int := 0;   // Настройка: Задержка отображения обрыва датчика
         Overflow_Delay : Int := 0;   // Настройка: Задержка отображения неисправности датчика
         StateHMI : Int;
         State : Word := 16#0;   // Выход: Состояние датчика
         Modeee : Word := 16#1;   // Настройка: Режим работы датчика
         bools : Word := 16#0;   // Все булевы параметры AI
         AI_RAW_MIN : Int := 0;   // Мин кода ацп
         AI_RAW_MAX : Int := 27648;   // Макс кода ацп
         Hihi_EN : Bool := false;   // Разрешение на сработку
         High_EN : Bool := false;   // Разрешение на сработку
         Low_En : Bool := false;   // Разрешение на сработку
         Lolo_EN : Bool := false;   // Разрешение на сработку
      END_STRUCT;
      AI_Config : Struct
         Hihi_Value : Real := 0.0;   // Уставка: Hihi
         High_Value : Real := 0.0;   // Уставка: High
         Low_Value : Real := 0.0;   // Уставка: Low
         Lolo_Value : Real := 0.0;   // Уставка: Lolo
         MIN_Current : Real := 0.0;   // Настройка: Минимальное входное значение тока
         MAX_Current : Real := 0.0;   // Настройка: Максимальное входное значение тока
         MAX_Value : Real := 0.0;   // Настройка: Максимальное значение измеряемой величины
         MIN_Value : Real := 0.0;   // Настройка: Минимальное значение измеряемой величины
         Underflow_RAW : Real := 0.0;   // Настройка: Значение кода ацп при обрыве
         Overflow_RAW : Real := 0.0;   // Настройка: Значение кода ацп при зашкале
         SCALED : Real := 0.0;   // Выход: Масштабированное в инженерные единицы значение входного сигнала
         ING_Value : Real := 0.0;   // Выход: Токовое значение датчика
         Manual_Value : Real := 0.0;   // Значение, введенное вручную
         Alarm_Delay : Int := 0;   // Настройка: Задержка срабатывания аварий
         Warning_Delay : Int := 0;   // Настройка: Задержка срабатывания предупреждений
         AVG_Delay : Real := 0.0;   // Настройка: Зона нечувствительности
         Underflow_Delay : Int := 0;   // Настройка: Задержка отображения обрыва датчика
         Overflow_Delay : Int := 0;   // Настройка: Задержка отображения неисправности датчика
         StateHMI : Int;
         State : Word := 16#0;   // Выход: Состояние датчика
         Modeee : Word := 16#0;   // Настройка: Режим работы датчика
         bools : Word := 16#0;   // Все булевы параметры AI
         AI_RAW_MIN : Int := 0;   // Мин кода ацп
         AI_RAW_MAX : Int := 0;   // Макс кода ацп
         Hihi_EN : Bool := false;   // Разрешение на сработку
         High_EN : Bool := false;   // Разрешение на сработку
         Low_En : Bool := false;   // Разрешение на сработку
         Lolo_EN : Bool := false;   // Разрешение на сработку
      END_STRUCT;
      ai_test : Int;
      DI_1_0 : Struct   // Сигнализатор уровня min
         Time_ON : Int := 0;   // Время перехода OFF->ON
         Time_OFF : Int := 0;   // Время перехода ON->OFF
         Input : Bool := false;   // Значение с модуля
         Disable : Bool := false;   // Запрет обработки канала
         Invert : Bool := false;   // Инертирование канала
         Output : Bool := false;   // Значение канала для логики
      END_STRUCT;
      DI_1_1 : Struct   // Сигнализатор уровня max
         Time_ON : Int := 0;   // Время перехода OFF->ON
         Time_OFF : Int := 0;   // Время перехода ON->OFF
         Input : Bool := false;   // Значение с модуля
         Disable : Bool := false;   // Запрет обработки канала
         Invert : Bool := false;   // Инертирование канала
         Output : Bool := false;   // Значение канала для логики
      END_STRUCT;
      DI_1_2 : Struct   // Клапан 1
         Time_ON : Int := 0;   // Время перехода OFF->ON
         Time_OFF : Int := 0;   // Время перехода ON->OFF
         Input : Bool := false;   // Значение с модуля
         Disable : Bool := false;   // Запрет обработки канала
         Invert : Bool := false;   // Инертирование канала
         Output : Bool := false;   // Значение канала для логики
      END_STRUCT;
      DI_1_3 : Struct   // Клапан 2
         Time_ON : Int := 0;   // Время перехода OFF->ON
         Time_OFF : Int := 0;   // Время перехода ON->OFF
         Input : Bool := false;   // Значение с модуля
         Disable : Bool := false;   // Запрет обработки канала
         Invert : Bool := false;   // Инертирование канала
         Output : Bool := false;   // Значение канала для логики
      END_STRUCT;
      DI_1_4 : Struct   // Резерв
         Time_ON : Int := 0;   // Время перехода OFF->ON
         Time_OFF : Int := 0;   // Время перехода ON->OFF
         Input : Bool := false;   // Значение с модуля
         Disable : Bool := false;   // Запрет обработки канала
         Invert : Bool := false;   // Инертирование канала
         Output : Bool := false;   // Значение канала для логики
      END_STRUCT;
      DI_1_5 : Struct   // Резерв
         Time_ON : Int := 0;   // Время перехода OFF->ON
         Time_OFF : Int := 0;   // Время перехода ON->OFF
         Input : Bool := false;   // Значение с модуля
         Disable : Bool := false;   // Запрет обработки канала
         Invert : Bool := false;   // Инертирование канала
         Output : Bool := false;   // Значение канала для логики
      END_STRUCT;
      DI_1_6 : Struct   // Работа горелки
         Time_ON : Int := 0;   // Время перехода OFF->ON
         Time_OFF : Int := 0;   // Время перехода ON->OFF
         Input : Bool := false;   // Значение с модуля
         Disable : Bool := false;   // Запрет обработки канала
         Invert : Bool := false;   // Инертирование канала
         Output : Bool := false;   // Значение канала для логики
      END_STRUCT;
      DI_1_7 : Struct   // Авария горелки
         Time_ON : Int := 0;   // Время перехода OFF->ON
         Time_OFF : Int := 0;   // Время перехода ON->OFF
         Input : Bool := false;   // Значение с модуля
         Disable : Bool := false;   // Запрет обработки канала
         Invert : Bool := false;   // Инертирование канала
         Output : Bool := false;   // Значение канала для логики
      END_STRUCT;
      DI_1_8 : Struct   // Резерв
         Time_ON : Int := 0;   // Время перехода OFF->ON
         Time_OFF : Int := 0;   // Время перехода ON->OFF
         Input : Bool := false;   // Значение с модуля
         Disable : Bool := false;   // Запрет обработки канала
         Invert : Bool := false;   // Инертирование канала
         Output : Bool := false;   // Значение канала для логики
      END_STRUCT;
      DI_1_9 : Struct   // Резерв
         Time_ON : Int := 0;   // Время перехода OFF->ON
         Time_OFF : Int := 0;   // Время перехода ON->OFF
         Input : Bool := false;   // Значение с модуля
         Disable : Bool := false;   // Запрет обработки канала
         Invert : Bool := false;   // Инертирование канала
         Output : Bool := false;   // Значение канала для логики
      END_STRUCT;
      DI_1_10 : Struct   // Резерв
         Time_ON : Int := 0;   // Время перехода OFF->ON
         Time_OFF : Int := 0;   // Время перехода ON->OFF
         Input : Bool := false;   // Значение с модуля
         Disable : Bool := false;   // Запрет обработки канала
         Invert : Bool := false;   // Инертирование канала
         Output : Bool := false;   // Значение канала для логики
      END_STRUCT;
      DI_1_11 : Struct   // Резерв
         Time_ON : Int := 0;   // Время перехода OFF->ON
         Time_OFF : Int := 0;   // Время перехода ON->OFF
         Input : Bool := false;   // Значение с модуля
         Disable : Bool := false;   // Запрет обработки канала
         Invert : Bool := false;   // Инертирование канала
         Output : Bool := false;   // Значение канала для логики
      END_STRUCT;
      DI_1_12 : Struct   // Резерв
         Time_ON : Int := 0;   // Время перехода OFF->ON
         Time_OFF : Int := 0;   // Время перехода ON->OFF
         Input : Bool := false;   // Значение с модуля
         Disable : Bool := false;   // Запрет обработки канала
         Invert : Bool := false;   // Инертирование канала
         Output : Bool := false;   // Значение канала для логики
      END_STRUCT;
      DI_1_13 : Struct   // Резерв
         Time_ON : Int := 0;   // Время перехода OFF->ON
         Time_OFF : Int := 0;   // Время перехода ON->OFF
         Input : Bool := false;   // Значение с модуля
         Disable : Bool := false;   // Запрет обработки канала
         Invert : Bool := false;   // Инертирование канала
         Output : Bool := false;   // Значение канала для логики
      END_STRUCT;
      DI_2_0 : Struct
         Time_ON : Int := 0;   // Время перехода OFF->ON
         Time_OFF : Int := 0;   // Время перехода ON->OFF
         Input : Bool := false;   // Значение с модуля
         Disable : Bool := false;   // Запрет обработки канала
         Invert : Bool := false;   // Инертирование канала
         Output : Bool := false;   // Значение канала для логики
      END_STRUCT;
      DI_2_1 : Struct
         Time_ON : Int := 0;   // Время перехода OFF->ON
         Time_OFF : Int := 0;   // Время перехода ON->OFF
         Input : Bool := false;   // Значение с модуля
         Disable : Bool := false;   // Запрет обработки канала
         Invert : Bool := false;   // Инертирование канала
         Output : Bool := false;   // Значение канала для логики
      END_STRUCT;
      DI_2_2 : Struct
         Time_ON : Int := 0;   // Время перехода OFF->ON
         Time_OFF : Int := 0;   // Время перехода ON->OFF
         Input : Bool := false;   // Значение с модуля
         Disable : Bool := false;   // Запрет обработки канала
         Invert : Bool := false;   // Инертирование канала
         Output : Bool := false;   // Значение канала для логики
      END_STRUCT;
      DI_2_3 : Struct
         Time_ON : Int := 0;   // Время перехода OFF->ON
         Time_OFF : Int := 0;   // Время перехода ON->OFF
         Input : Bool := false;   // Значение с модуля
         Disable : Bool := false;   // Запрет обработки канала
         Invert : Bool := false;   // Инертирование канала
         Output : Bool := false;   // Значение канала для логики
      END_STRUCT;
      DI_2_4 : Struct
         Time_ON : Int := 0;   // Время перехода OFF->ON
         Time_OFF : Int := 0;   // Время перехода ON->OFF
         Input : Bool := false;   // Значение с модуля
         Disable : Bool := false;   // Запрет обработки канала
         Invert : Bool := false;   // Инертирование канала
         Output : Bool := false;   // Значение канала для логики
      END_STRUCT;
      DI_2_5 : Struct
         Time_ON : Int := 0;   // Время перехода OFF->ON
         Time_OFF : Int := 0;   // Время перехода ON->OFF
         Input : Bool := false;   // Значение с модуля
         Disable : Bool := false;   // Запрет обработки канала
         Invert : Bool := false;   // Инертирование канала
         Output : Bool := false;   // Значение канала для логики
      END_STRUCT;
      DI_2_6 : Struct
         Time_ON : Int := 0;   // Время перехода OFF->ON
         Time_OFF : Int := 0;   // Время перехода ON->OFF
         Input : Bool := false;   // Значение с модуля
         Disable : Bool := false;   // Запрет обработки канала
         Invert : Bool := false;   // Инертирование канала
         Output : Bool := false;   // Значение канала для логики
      END_STRUCT;
      DI_2_7 : Struct
         Time_ON : Int := 0;   // Время перехода OFF->ON
         Time_OFF : Int := 0;   // Время перехода ON->OFF
         Input : Bool := false;   // Значение с модуля
         Disable : Bool := false;   // Запрет обработки канала
         Invert : Bool := false;   // Инертирование канала
         Output : Bool := false;   // Значение канала для логики
      END_STRUCT;
      DI_2_8 : Struct
         Time_ON : Int := 0;   // Время перехода OFF->ON
         Time_OFF : Int := 0;   // Время перехода ON->OFF
         Input : Bool := false;   // Значение с модуля
         Disable : Bool := false;   // Запрет обработки канала
         Invert : Bool := false;   // Инертирование канала
         Output : Bool := false;   // Значение канала для логики
      END_STRUCT;
      DI_2_9 : Struct
         Time_ON : Int := 0;   // Время перехода OFF->ON
         Time_OFF : Int := 0;   // Время перехода ON->OFF
         Input : Bool := false;   // Значение с модуля
         Disable : Bool := false;   // Запрет обработки канала
         Invert : Bool := false;   // Инертирование канала
         Output : Bool := false;   // Значение канала для логики
      END_STRUCT;
      DI_2_10 : Struct
         Time_ON : Int := 0;   // Время перехода OFF->ON
         Time_OFF : Int := 0;   // Время перехода ON->OFF
         Input : Bool := false;   // Значение с модуля
         Disable : Bool := false;   // Запрет обработки канала
         Invert : Bool := false;   // Инертирование канала
         Output : Bool := false;   // Значение канала для логики
      END_STRUCT;
      DI_2_11 : Struct
         Time_ON : Int := 0;   // Время перехода OFF->ON
         Time_OFF : Int := 0;   // Время перехода ON->OFF
         Input : Bool := false;   // Значение с модуля
         Disable : Bool := false;   // Запрет обработки канала
         Invert : Bool := false;   // Инертирование канала
         Output : Bool := false;   // Значение канала для логики
      END_STRUCT;
      DI_2_12 : Struct
         Time_ON : Int := 0;   // Время перехода OFF->ON
         Time_OFF : Int := 0;   // Время перехода ON->OFF
         Input : Bool := false;   // Значение с модуля
         Disable : Bool := false;   // Запрет обработки канала
         Invert : Bool := false;   // Инертирование канала
         Output : Bool := false;   // Значение канала для логики
      END_STRUCT;
      DI_2_13 : Struct
         Time_ON : Int := 0;   // Время перехода OFF->ON
         Time_OFF : Int := 0;   // Время перехода ON->OFF
         Input : Bool := false;   // Значение с модуля
         Disable : Bool := false;   // Запрет обработки канала
         Invert : Bool := false;   // Инертирование канала
         Output : Bool := false;   // Значение канала для логики
      END_STRUCT;
      DI_2_14 : Struct
         Time_ON : Int := 0;   // Время перехода OFF->ON
         Time_OFF : Int := 0;   // Время перехода ON->OFF
         Input : Bool := false;   // Значение с модуля
         Disable : Bool := false;   // Запрет обработки канала
         Invert : Bool := false;   // Инертирование канала
         Output : Bool := false;   // Значение канала для логики
      END_STRUCT;
      DI_2_15 : Struct
         Time_ON : Int := 0;   // Время перехода OFF->ON
         Time_OFF : Int := 0;   // Время перехода ON->OFF
         Input : Bool := false;   // Значение с модуля
         Disable : Bool := false;   // Запрет обработки канала
         Invert : Bool := false;   // Инертирование канала
         Output : Bool := false;   // Значение канала для логики
      END_STRUCT;
      DO_1_0 : Struct   // ПАСВ светозвуковой
         Time_ON : Int := 0;   // Время перехода OFF->ON
         Time_OFF : Int := 0;   // Время перехода ON->OFF
         Input : Bool := false;   // Значение от логики
         Disable : Bool := false;   // Запрет обработки канала
         Invert : Bool := false;   // Инертирование канала
         Output : Bool := false;   // Значение на модуль
      END_STRUCT;
      DO_1_1 : Struct   // ПАСВ светозвуковой
         Time_ON : Int := 0;   // Время перехода OFF->ON
         Time_OFF : Int := 0;   // Время перехода ON->OFF
         Input : Bool := false;   // Значение от логики
         Disable : Bool := false;   // Запрет обработки канала
         Invert : Bool := false;   // Инертирование канала
         Output : Bool := false;   // Значение на модуль
      END_STRUCT;
      DO_1_2 : Struct   // Пуск/стоп горелки
         Time_ON : Int := 0;   // Время перехода OFF->ON
         Time_OFF : Int := 0;   // Время перехода ON->OFF
         Input : Bool := false;   // Значение от логики
         Disable : Bool := false;   // Запрет обработки канала
         Invert : Bool := false;   // Инертирование канала
         Output : Bool := false;   // Значение на модуль
      END_STRUCT;
      DO_1_3 : Struct   // Клапан 1
         Time_ON : Int := 0;   // Время перехода OFF->ON
         Time_OFF : Int := 0;   // Время перехода ON->OFF
         Input : Bool := false;   // Значение от логики
         Disable : Bool := false;   // Запрет обработки канала
         Invert : Bool := false;   // Инертирование канала
         Output : Bool := false;   // Значение на модуль
      END_STRUCT;
      DO_1_4 : Struct   // Клапан 2
         Time_ON : Int := 0;   // Время перехода OFF->ON
         Time_OFF : Int := 0;   // Время перехода ON->OFF
         Input : Bool := false;   // Значение от логики
         Disable : Bool := false;   // Запрет обработки канала
         Invert : Bool := false;   // Инертирование канала
         Output : Bool := false;   // Значение на модуль
      END_STRUCT;
      DO_1_5 : Struct   // ИВНТР
         Time_ON : Int := 0;   // Время перехода OFF->ON
         Time_OFF : Int := 0;   // Время перехода ON->OFF
         Input : Bool := false;   // Значение от логики
         Disable : Bool := false;   // Запрет обработки канала
         Invert : Bool := false;   // Инертирование канала
         Output : Bool := false;   // Значение на модуль
      END_STRUCT;
      DO_1_6 : Struct   // Резерв
         Time_ON : Int := 0;   // Время перехода OFF->ON
         Time_OFF : Int := 0;   // Время перехода ON->OFF
         Input : Bool := false;   // Значение от логики
         Disable : Bool := false;   // Запрет обработки канала
         Invert : Bool := false;   // Инертирование канала
         Output : Bool := false;   // Значение на модуль
      END_STRUCT;
      DO_1_7 : Struct   // Резерв
         Time_ON : Int := 0;   // Время перехода OFF->ON
         Time_OFF : Int := 0;   // Время перехода ON->OFF
         Input : Bool := false;   // Значение от логики
         Disable : Bool := false;   // Запрет обработки канала
         Invert : Bool := false;   // Инертирование канала
         Output : Bool := false;   // Значение на модуль
      END_STRUCT;
      DO_1_8 : Struct   // Резерв
         Time_ON : Int := 0;   // Время перехода OFF->ON
         Time_OFF : Int := 0;   // Время перехода ON->OFF
         Input : Bool := false;   // Значение от логики
         Disable : Bool := false;   // Запрет обработки канала
         Invert : Bool := false;   // Инертирование канала
         Output : Bool := false;   // Значение на модуль
      END_STRUCT;
      DO_2_0 : Struct   // Резерв
         Time_ON : Int := 0;   // Время перехода OFF->ON
         Time_OFF : Int := 0;   // Время перехода ON->OFF
         Input : Bool := false;   // Значение от логики
         Disable : Bool := false;   // Запрет обработки канала
         Invert : Bool := false;   // Инертирование канала
         Output : Bool := false;   // Значение на модуль
      END_STRUCT;
      DO_2_1 : Struct
         Time_ON : Int := 0;   // Время перехода OFF->ON
         Time_OFF : Int := 0;   // Время перехода ON->OFF
         Input : Bool := false;   // Значение от логики
         Disable : Bool := false;   // Запрет обработки канала
         Invert : Bool := false;   // Инертирование канала
         Output : Bool := false;   // Значение на модуль
      END_STRUCT;
      DO_2_2 : Struct
         Time_ON : Int := 0;   // Время перехода OFF->ON
         Time_OFF : Int := 0;   // Время перехода ON->OFF
         Input : Bool := false;   // Значение от логики
         Disable : Bool := false;   // Запрет обработки канала
         Invert : Bool := false;   // Инертирование канала
         Output : Bool := false;   // Значение на модуль
      END_STRUCT;
      DO_2_3 : Struct
         Time_ON : Int := 0;   // Время перехода OFF->ON
         Time_OFF : Int := 0;   // Время перехода ON->OFF
         Input : Bool := false;   // Значение от логики
         Disable : Bool := false;   // Запрет обработки канала
         Invert : Bool := false;   // Инертирование канала
         Output : Bool := false;   // Значение на модуль
      END_STRUCT;
      Channel_Number : Int;
      Read : Bool;
      Write : Bool;
      GAZ_State : Int;
      CH_NUMBER : Array[0..20] of Bool;
   END_VAR
BEGIN
END_DATA_BLOCK

DATA_BLOCK "PMP_DB"   // DB2
{ S7_Optimized_Access := 'FALSE' }
VERSION : 0.1
   VAR
      Burner : Struct
         State : Int;
         CMD_in : Int;
         Alarm : Int;
      END_STRUCT;
      Valve_oil_in : Struct
         State : Int;
         State_ctrl : Bool;
         Alarm : Int;
         Cmd_in : Int;
         Cmd_out : Bool;
         bools : Int;
         Deblock : Bool;
      END_STRUCT;
      Valve_oil_out : Struct
         State : Int;
         State_ctrl : Bool;
         Alarm : Int;
         Cmd_in : Int;
         Cmd_out : Bool;
         bools : Int;
         Deblock : Bool;
      END_STRUCT;
      Valve_gaz_in : Struct
         State : Int;
         State_ctrl : Bool;
         Alarm : Int;
         Cmd_in : Int;
         Cmd_out : Bool;
         bools : Int;
         Deblock : Bool;
      END_STRUCT;
      Valve_ctrl : Struct
         State : Int;
         Cmd_in : Int;
         TIME_shod : Int;
         TIME_hod : Int;
         bools : DWord;
      END_STRUCT;
      Vent_work_timer : Bool;
      Vent_work_timer_stoped : Bool;
      Hiter_BT : Struct
         Mode : Bool;
         T_state : Int;
         CMD : Bool;
         Avar_stop : Bool;
      END_STRUCT;
      MB_CTRL_EN : Bool;   // Разрешение управлния с телемеханики
      baud_rate : UDInt := 9600;   // MB скорость
      MB_addr : UInt := 1;   // MB адрес
      BDR_OFF_RST : Bool;   // Сброс расцепителя "Отключить БДР"
   END_VAR
BEGIN
END_DATA_BLOCK

DATA_BLOCK "Slave"   // DB16
{ S7_Optimized_Access := 'FALSE' }
VERSION : 0.1
   VAR
      MBVerh_0 : Int;   // Давление на выкиде НД1, МПа PT1
      MBVerh_1 : Int;   // Давление на выкиде НД2, МПа PT2
      MBVerh_2 : Int;   // Температура в БТ, С ТТ1
      MBVerh_3 : Int;
      MBVerh_4 : Int;   // Перепад давления на фильтре 1, МПа РТ3
      MBVerh_5 : Int;   // Перепад давления на фильтре 2, МПа РТ4
      MBVerh_6 : Int;   // Температура в емкости Б1, С ТТ3
      MBVerh_7 : Int;   // Температура в емкости Б1, С ТТ3
      MBVerh_8 : Int;   // Уровень в емкости Б1, см LT1
      MBVerh_9 : Int;   // Расход, м3/ч FT1
      MBVerh_10 : Int;
      MBVerh_11 : Int;
      MBVerh_12 : Int;   // Разрешить откл БДР по пожару
      MBVerh_13 : Int;
      MBVerh_14 : Int;
      MBVerh_15 : Int;
      MBVerh_16 : Int;
      Burner_State : Word;
      T_Need_Emk : Int;   // Максимальная температура в теплоносители
      T_Need_Oil : Int;   // Максимальная температура нефти
      T_Lo : Int;   // Минимальаня температура для автопуска
      T_Time_ON : Int;   // Время включения большого горения в минутах
      T_Need_Big_Gorenie : Real;   // Если не дошло до уставки для включения большого горения
      T_Need_Emk_TM : Int;   // Максимальная температура в теплоносители
      T_Need_Oil_TM : Int;   // Максимальная температура нефти
      T_Lo_TM : Int;   // Минимальаня температура для автопуска
      T_Time_ON_TM : Int;   // Время включения большого горения в минутах
      T_Need_Big_Gorenie_TM : Real;   // Если не дошло до уставки для включения большого горения
      CMD_TM : Int;
      State_1 : Int;
      State_2 : Int;
      State_3 : Int;
   END_VAR
BEGIN
END_DATA_BLOCK

DATA_BLOCK "MB_Diagnostic"   // DB19
{ S7_Optimized_Access := 'FALSE' }
VERSION : 0.1
   VAR
      comm_done : Bool;
      comm_er : Bool;
      comm_sr : Word;
      slave_er : Bool;
      slave_st : Word;
   END_VAR
BEGIN
END_DATA_BLOCK

DATA_BLOCK "DB_TST"   // DB33
{ S7_Optimized_Access := 'FALSE' }
VERSION : 0.1
   VAR
      CH_NUMBER : Int;
      CH_NUMBER_OLD : Int;
      AI : Struct   // Структура AI
         Hihi_Value : Real := 70.0;   // Уставка: Hihi
         High_Value : Real := 60.0;   // Уставка: High
         Low_Value : Real := 30.0;   // Уставка: Low
         Lolo_Value : Real := 20.0;   // Уставка: Lolo
         MIN_Current : Real := 4.0;   // Настройка: Минимальное входное значение тока
         MAX_Current : Real := 20.0;   // Настройка: Максимальное входное значение тока
         MAX_Value : Real := 100.0;   // Настройка: Максимальное значение измеряемой величины
         MIN_Value : Real := 0.0;   // Настройка: Минимальное значение измеряемой величины
         Underflow_RAW : Real := -10.0;   // Настройка: Значение кода ацп при обрыве
         Overflow_RAW : Real := 27650.0;   // Настройка: Значение кода ацп при зашкале
         SCALED : Real;   // Выход: Масштабированное в инженерные единицы значение входного сигнала
         ING_Value : Real;   // Выход: Токовое значение датчика
         Manual_Value : Real := 50.0;   // Значение, введенное вручную
         Alarm_Delay : Int;   // Настройка: Задержка срабатывания аварий
         Warning_Delay : Int;   // Настройка: Задержка срабатывания предупреждений
         AVG_Delay : Real;   // Настройка: Зона нечувствительности
         Underflow_Delay : Int;   // Настройка: Задержка отображения обрыва датчика
         Overflow_Delay : Int;   // Настройка: Задержка отображения неисправности датчика
         State : Word;   // Выход: Состояние датчика
         Modeee : Word := 16#1;   // Настройка: Режим работы датчика
         bools : Word;   // Все булевы параметры AI
         AI_RAW_MIN : Int := 0;   // Мин кода ацп
         AI_RAW_MAX : Int := 27648;   // Макс кода ацп
         Hihi_EN : Bool;   // Разрешение на сработку
         High_EN : Bool;   // Разрешение на сработку
         Low_En : Bool;   // Разрешение на сработку
         Lolo_EN : Bool;   // Разрешение на сработку
      END_STRUCT;
      AI_RAW : Int;
      TST_State : Bool;
      TST_State_Pusk : Bool;
      Valve_opening : Bool;
      Valve_closing : Bool;
      Valve_Pos : Struct   // Аналоговый датчик положения клапана
         Hihi_Value : Real;   // Уставка: Hihi
         High_Value : Real;   // Уставка: High
         Low_Value : Real;   // Уставка: Low
         Lolo_Value : Real;   // Уставка: Lolo
         MIN_Current : Real;   // Настройка: Минимальное входное значение тока
         MAX_Current : Real;   // Настройка: Максимальное входное значение тока
         MAX_Value : Real;   // Настройка: Максимальное значение измеряемой величины
         MIN_Value : Real;   // Настройка: Минимальное значение измеряемой величины
         Underflow_RAW : Real;   // Настройка: Значение кода ацп при обрыве
         Overflow_RAW : Real;   // Настройка: Значение кода ацп при зашкале
         SCALED : Real;   // Выход: Масштабированное в инженерные единицы значение входного сигнала
         ING_Value : Real;   // Выход: Токовое значение датчика
         Manual_Value : Real;   // Значение, введенное вручную
         Alarm_Delay : Int;   // Настройка: Задержка срабатывания аварий
         Warning_Delay : Int;   // Настройка: Задержка срабатывания предупреждений
         AVG_Delay : Real;   // Настройка: Зона нечувствительности
         Underflow_Delay : Int;   // Настройка: Задержка отображения обрыва датчика
         Overflow_Delay : Int;   // Настройка: Задержка отображения неисправности датчика
         State : Word;   // Выход: Состояние датчика
         Modeee : Word;   // Настройка: Режим работы датчика
         bools : Word;   // Все булевы параметры AI
         AI_RAW_MIN : Int;   // Мин кода ацп
         AI_RAW_MAX : Int;   // Макс кода ацп
         Hihi_EN : Bool;   // Разрешение на сработку
         High_EN : Bool;   // Разрешение на сработку
         Low_En : Bool;   // Разрешение на сработку
         Lolo_EN : Bool;   // Разрешение на сработку
      END_STRUCT;
      CMD_Open_Out : Bool;
      CMD_Close_Out : Bool;
      Burner : Struct
         State_W : DWord;
         State : Int;
         CMD_Start : Bool;
         CMD_Stop : Bool;
         CMD_RST_Alarm : Bool;
         CMD_Start_Stop : Bool;
         Alarm_W : DWord;
         Alarm_INT : Int;
         Alarm : Bool;
         Auto_Pause : Bool;
         Flag_Auto_Pause : Bool;
         Fire : Bool;
         mode_Hmi : Bool;
         mode_ARM : Bool;
         mode : Bool;
         ARM_start : Bool;
         ARM_stop : Bool;
         ARM_deblock : Bool;
      END_STRUCT;
      Max_Open : Real := 50.0;
      TST_Journey : Word;
      "a" : Bool;
      a1 : Bool;
      "b" : Bool;
      c : Bool;
      d : Bool;
      "e" : Bool;
      T_Need_Emk_Hi : Real := 80.0;   // Максимальная температура в теплоносители
      T_Need_Oil_Hi : Real := 55.0;   // Максимальная температура нефти
      T_Lo_TM : Real := 30.0;   // Минимальаня температура для автопуска
      CMD_TM : Int;
      T_Time_ON : Int := 30;   // Время включения большого горения в минутах
      T_Need_Big_Gorenie : Real := 30.0;   // Если не дошло до уставки для включения большого горения
      T_Time_ON_TM : Int := 30;   // Время включения большого горения в минутах
      T_Need_Big_Gorenie_TM : Real;   // Если не дошло до уставки для включения большого горения
      Need_open_cl_1 : Bool;   // Открыть клапан на запальную горелку
      Need_open_cl_2 : Bool;   // Открыть клапан на основную горелку
      Valve_alarm_1 : Bool;   // Аврия запальной горелки
      Valve_alarm_2 : Bool;   // Авария основной горелки
      Valve_1 : Struct
         CMD_Open : Bool;   // Команда открыть
         CMD_Close : Bool;   // Команда закрыть
         CMD_ALRM_Stop : Bool;
         State : Word;
         State_INT : Int;
         Mode : Bool;   // 0-ручной, 1-авто
         Alarm : Word;
         bools : Word;
         RST_ALRM : Bool;
         CMD_Open_Out : Bool;   // управление открыть
         CMD_Close_Out : Bool;   // управление закрыть
      END_STRUCT;
      Valve_2 : Struct
         CMD_Open : Bool;   // Команда открыть
         CMD_Close : Bool;   // Команда закрыть
         CMD_ALRM_Stop : Bool;
         State : Word;
         State_INT : Int;
         Mode : Bool;   // 0-ручной, 1-авто
         Alarm : Word;
         bools : Word;
         RST_ALRM : Bool;
         CMD_Open_Out : Bool;   // управление открыть
         CMD_Close_Out : Bool;   // управление закрыть
      END_STRUCT;
      RST_alarm_burner : Bool;
      Gaz_state : Int;   // Состояние газоанализатора
      T_Emk_Lo_Hmi : Real;
      T_Emk_Hi_Hmi : Real;
      T_Oil_Lo_Hmi : Real;
      T_Oil_Hi_Hmi : Real;
      Gaz_porog1 : Bool;
      Gaz_porog2 : Bool;
      Gaz_neispravnost : Bool;
      P_gaz_out : Struct
         Hihi : Bool;
         Hi : Bool;
         Lo : Bool;
         Lolo : Bool;
      END_STRUCT;
      P_gaz_in : Struct
         Hihi : Bool;
         Hi : Bool;
         Lo : Bool;
         Lolo : Bool;
      END_STRUCT;
      P_gaza : Struct
         Hihi : Bool;
         Hi : Bool;
         Lo : Bool;
         Lolo : Bool;
      END_STRUCT;
      T_gaza_out : Struct
         Hihi : Bool;
         Hi : Bool;
         Lo : Bool;
         Lolo : Bool;
      END_STRUCT;
      T_dym_gazov : Struct
         Hihi : Bool;
         Hi : Bool;
         Lo : Bool;
         Lolo : Bool;
      END_STRUCT;
      T_emk : Struct
         Hihi : Bool;
         Hi : Bool;
         Lo : Bool;
         Lolo : Bool;
      END_STRUCT;
      T_emk_B1 : Struct
         Hihi : Bool;
         Hi : Bool;
         Lo : Bool;
         Lolo : Bool;
      END_STRUCT;
      Gazik : Struct
         Hihi : Bool;
         Hi : Bool;
         Lo : Bool;
         Lolo : Bool;
      END_STRUCT;
      Delay_produv : Int := 10;
      Fire_interval : Int := 5;
      Fire_delay : Int := 5;
      Open_cl2_delay : Int := 5;
   END_VAR
BEGIN
END_DATA_BLOCK

// folder: System blocks/Program resources

DATA_BLOCK "Time_Opening_cl_1"   // DB3
{ S7_Optimized_Access := 'TRUE' }
AUTHOR : Simatic
FAMILY : IEC
NAME : IEC_TMR
VERSION : 1.0
// stored: InstanceOfName IEC_TIMER
"IEC_TIMER"
BEGIN
END_DATA_BLOCK

DATA_BLOCK "Time_Closing_cl_2"   // DB4
{ S7_Optimized_Access := 'TRUE' }
AUTHOR : Simatic
FAMILY : IEC
NAME : IEC_TMR
VERSION : 1.0
// stored: InstanceOfName IEC_TIMER
"IEC_TIMER"
BEGIN
END_DATA_BLOCK

DATA_BLOCK "AI_3_4_Hihi_Timer"   // DB5
{ S7_Optimized_Access := 'TRUE' }
AUTHOR : Simatic
FAMILY : IEC
NAME : IEC_TMR
VERSION : 1.0
// stored: InstanceOfName IEC_TIMER
"IEC_TIMER"
BEGIN
END_DATA_BLOCK

DATA_BLOCK "DI_1_0_TON"   // DB6
{ S7_Optimized_Access := 'TRUE' }
AUTHOR : Simatic
FAMILY : IEC
NAME : IEC_TMR
VERSION : 1.0
// stored: InstanceOfName IEC_TIMER
"IEC_TIMER"
BEGIN
END_DATA_BLOCK

DATA_BLOCK "DI_1_0_TOF"   // DB7
{ S7_Optimized_Access := 'TRUE' }
AUTHOR : Simatic
FAMILY : IEC
NAME : IEC_TMR
VERSION : 1.0
// stored: InstanceOfName IEC_TIMER
"IEC_TIMER"
BEGIN
END_DATA_BLOCK

DATA_BLOCK "DI_1_1_TON"   // DB8
{ S7_Optimized_Access := 'TRUE' }
AUTHOR : Simatic
FAMILY : IEC
NAME : IEC_TMR
VERSION : 1.0
// stored: InstanceOfName IEC_TIMER
"IEC_TIMER"
BEGIN
END_DATA_BLOCK

DATA_BLOCK "Timer_need_cl_2"   // DB9
{ S7_Optimized_Access := 'TRUE' }
AUTHOR : Simatic
FAMILY : IEC
NAME : IEC_TMR
VERSION : 1.0
// stored: InstanceOfName IEC_TIMER
"IEC_TIMER"
BEGIN
END_DATA_BLOCK

DATA_BLOCK "DI_1_2_TON"   // DB10
{ S7_Optimized_Access := 'TRUE' }
AUTHOR : Simatic
FAMILY : IEC
NAME : IEC_TMR
VERSION : 1.0
// stored: InstanceOfName IEC_TIMER
"IEC_TIMER"
BEGIN
END_DATA_BLOCK

DATA_BLOCK "Burner_Fire_Timer"   // DB12
{ S7_Optimized_Access := 'TRUE' }
AUTHOR : Simatic
FAMILY : IEC
NAME : IEC_TMR
VERSION : 1.0
// stored: InstanceOfName IEC_TIMER
"IEC_TIMER"
BEGIN
END_DATA_BLOCK

DATA_BLOCK "Burner_Fire_Timer_Delay"   // DB13
{ S7_Optimized_Access := 'TRUE' }
AUTHOR : Simatic
FAMILY : IEC
NAME : IEC_TMR
VERSION : 1.0
// stored: InstanceOfName IEC_TIMER
"IEC_TIMER"
BEGIN
END_DATA_BLOCK

DATA_BLOCK "Start_Fire_Counter"   // DB14
{ S7_Optimized_Access := 'TRUE' }
AUTHOR : Simatic
FAMILY : IEC
NAME : CNTR
VERSION : 1.0
// stored: InstanceOfName IEC_COUNTER
"IEC_COUNTER"
BEGIN
END_DATA_BLOCK

DATA_BLOCK "Delay_produv"   // DB17
{ S7_Optimized_Access := 'TRUE' }
AUTHOR : Simatic
FAMILY : IEC
NAME : IEC_TMR
VERSION : 1.0
// stored: InstanceOfName IEC_TIMER
"IEC_TIMER"
BEGIN
END_DATA_BLOCK

DATA_BLOCK "IEC_Timer_0_DB"   // DB18
{ S7_Optimized_Access := 'TRUE' }
AUTHOR : Simatic
FAMILY : IEC
NAME : IEC_TMR
VERSION : 1.0
// stored: InstanceOfName IEC_TIMER
"IEC_TIMER"
BEGIN
END_DATA_BLOCK

DATA_BLOCK "AI_3_2_Hihi_Timer"   // DB20
{ S7_Optimized_Access := 'TRUE' }
AUTHOR : Simatic
FAMILY : IEC
NAME : IEC_TMR
VERSION : 1.0
// stored: InstanceOfName IEC_TIMER
"IEC_TIMER"
BEGIN
END_DATA_BLOCK

DATA_BLOCK "AI_3_5_Hihi_Timer"   // DB21
{ S7_Optimized_Access := 'TRUE' }
AUTHOR : Simatic
FAMILY : IEC
NAME : IEC_TMR
VERSION : 1.0
// stored: InstanceOfName IEC_TIMER
"IEC_TIMER"
BEGIN
END_DATA_BLOCK

DATA_BLOCK "AI_3_7_Hihi_Timer"   // DB22
{ S7_Optimized_Access := 'TRUE' }
AUTHOR : Simatic
FAMILY : IEC
NAME : IEC_TMR
VERSION : 1.0
// stored: InstanceOfName IEC_TIMER
"IEC_TIMER"
BEGIN
END_DATA_BLOCK

DATA_BLOCK "AI_2_0_Hihi_Timer"   // DB23
{ S7_Optimized_Access := 'TRUE' }
AUTHOR : Simatic
FAMILY : IEC
NAME : IEC_TMR
VERSION : 1.0
// stored: InstanceOfName IEC_TIMER
"IEC_TIMER"
BEGIN
END_DATA_BLOCK

DATA_BLOCK "AI_3_6_Hihi_Timer"   // DB24
{ S7_Optimized_Access := 'TRUE' }
AUTHOR : Simatic
FAMILY : IEC
NAME : IEC_TMR
VERSION : 1.0
// stored: InstanceOfName IEC_TIMER
"IEC_TIMER"
BEGIN
END_DATA_BLOCK

DATA_BLOCK "AI_3_3_Hihi_Timer"   // DB25
{ S7_Optimized_Access := 'TRUE' }
AUTHOR : Simatic
FAMILY : IEC
NAME : IEC_TMR
VERSION : 1.0
// stored: InstanceOfName IEC_TIMER
"IEC_TIMER"
BEGIN
END_DATA_BLOCK

DATA_BLOCK "AI_3_2_High_Timer"   // DB26
{ S7_Optimized_Access := 'TRUE' }
AUTHOR : Simatic
FAMILY : IEC
NAME : IEC_TMR
VERSION : 1.0
// stored: InstanceOfName IEC_TIMER
"IEC_TIMER"
BEGIN
END_DATA_BLOCK

DATA_BLOCK "AI_3_5_High_Timer"   // DB27
{ S7_Optimized_Access := 'TRUE' }
AUTHOR : Simatic
FAMILY : IEC
NAME : IEC_TMR
VERSION : 1.0
// stored: InstanceOfName IEC_TIMER
"IEC_TIMER"
BEGIN
END_DATA_BLOCK

DATA_BLOCK "AI_3_3_High_Timer"   // DB28
{ S7_Optimized_Access := 'TRUE' }
AUTHOR : Simatic
FAMILY : IEC
NAME : IEC_TMR
VERSION : 1.0
// stored: InstanceOfName IEC_TIMER
"IEC_TIMER"
BEGIN
END_DATA_BLOCK

DATA_BLOCK "AI_3_4_High_Timer"   // DB29
{ S7_Optimized_Access := 'TRUE' }
AUTHOR : Simatic
FAMILY : IEC
NAME : IEC_TMR
VERSION : 1.0
// stored: InstanceOfName IEC_TIMER
"IEC_TIMER"
BEGIN
END_DATA_BLOCK

DATA_BLOCK "AI_2_0_High_Timer"   // DB32
{ S7_Optimized_Access := 'TRUE' }
AUTHOR : Simatic
FAMILY : IEC
NAME : IEC_TMR
VERSION : 1.0
// stored: InstanceOfName IEC_TIMER
"IEC_TIMER"
BEGIN
END_DATA_BLOCK

DATA_BLOCK "AI_3_7_High_Timer"   // DB34
{ S7_Optimized_Access := 'TRUE' }
AUTHOR : Simatic
FAMILY : IEC
NAME : IEC_TMR
VERSION : 1.0
// stored: InstanceOfName IEC_TIMER
"IEC_TIMER"
BEGIN
END_DATA_BLOCK

DATA_BLOCK "Time_Opening_cl_2"   // DB35
{ S7_Optimized_Access := 'TRUE' }
AUTHOR : Simatic
FAMILY : IEC
NAME : IEC_TMR
VERSION : 1.0
// stored: InstanceOfName IEC_TIMER
"IEC_TIMER"
BEGIN
END_DATA_BLOCK

DATA_BLOCK "Time_Closing_cl_1"   // DB36
{ S7_Optimized_Access := 'TRUE' }
AUTHOR : Simatic
FAMILY : IEC
NAME : IEC_TMR
VERSION : 1.0
// stored: InstanceOfName IEC_TIMER
"IEC_TIMER"
BEGIN
END_DATA_BLOCK

DATA_BLOCK "Timer_Not_Start"   // DB37
{ S7_Optimized_Access := 'TRUE' }
AUTHOR : Simatic
FAMILY : IEC
NAME : IEC_TMR
VERSION : 1.0
// stored: InstanceOfName IEC_TIMER
"IEC_TIMER"
BEGIN
END_DATA_BLOCK

DATA_BLOCK "AI_2_0_Low_Timer"   // DB38
{ S7_Optimized_Access := 'TRUE' }
AUTHOR : Simatic
FAMILY : IEC
NAME : IEC_TMR
VERSION : 1.0
// stored: InstanceOfName IEC_TIMER
"IEC_TIMER"
BEGIN
END_DATA_BLOCK

DATA_BLOCK "AI_3_6_High_Timer"   // DB40
{ S7_Optimized_Access := 'TRUE' }
AUTHOR : Simatic
FAMILY : IEC
NAME : IEC_TMR
VERSION : 1.0
// stored: InstanceOfName IEC_TIMER
"IEC_TIMER"
BEGIN
END_DATA_BLOCK

DATA_BLOCK "AI_3_5_Low_Timer"   // DB41
{ S7_Optimized_Access := 'TRUE' }
AUTHOR : Simatic
FAMILY : IEC
NAME : IEC_TMR
VERSION : 1.0
// stored: InstanceOfName IEC_TIMER
"IEC_TIMER"
BEGIN
END_DATA_BLOCK

DATA_BLOCK "AI_3_4_Low_Timer"   // DB42
{ S7_Optimized_Access := 'TRUE' }
AUTHOR : Simatic
FAMILY : IEC
NAME : IEC_TMR
VERSION : 1.0
// stored: InstanceOfName IEC_TIMER
"IEC_TIMER"
BEGIN
END_DATA_BLOCK

DATA_BLOCK "AI_3_3_Low_Timer"   // DB43
{ S7_Optimized_Access := 'TRUE' }
AUTHOR : Simatic
FAMILY : IEC
NAME : IEC_TMR
VERSION : 1.0
// stored: InstanceOfName IEC_TIMER
"IEC_TIMER"
BEGIN
END_DATA_BLOCK

DATA_BLOCK "AI_3_6_Low_Timer"   // DB44
{ S7_Optimized_Access := 'TRUE' }
AUTHOR : Simatic
FAMILY : IEC
NAME : IEC_TMR
VERSION : 1.0
// stored: InstanceOfName IEC_TIMER
"IEC_TIMER"
BEGIN
END_DATA_BLOCK

DATA_BLOCK "AI_3_2_Low_Timer"   // DB45
{ S7_Optimized_Access := 'TRUE' }
AUTHOR : Simatic
FAMILY : IEC
NAME : IEC_TMR
VERSION : 1.0
// stored: InstanceOfName IEC_TIMER
"IEC_TIMER"
BEGIN
END_DATA_BLOCK

DATA_BLOCK "AI_3_7_Low_Timer"   // DB46
{ S7_Optimized_Access := 'TRUE' }
AUTHOR : Simatic
FAMILY : IEC
NAME : IEC_TMR
VERSION : 1.0
// stored: InstanceOfName IEC_TIMER
"IEC_TIMER"
BEGIN
END_DATA_BLOCK

DATA_BLOCK "AI_2_0_Lolo_Timer"   // DB47
{ S7_Optimized_Access := 'TRUE' }
AUTHOR : Simatic
FAMILY : IEC
NAME : IEC_TMR
VERSION : 1.0
// stored: InstanceOfName IEC_TIMER
"IEC_TIMER"
BEGIN
END_DATA_BLOCK

DATA_BLOCK "AI_2_0_Overflow_Timer"   // DB48
{ S7_Optimized_Access := 'TRUE' }
AUTHOR : Simatic
FAMILY : IEC
NAME : IEC_TMR
VERSION : 1.0
// stored: InstanceOfName IEC_TIMER
"IEC_TIMER"
BEGIN
END_DATA_BLOCK

DATA_BLOCK "AI_2_0_WB_Timer"   // DB49
{ S7_Optimized_Access := 'TRUE' }
AUTHOR : Simatic
FAMILY : IEC
NAME : IEC_TMR
VERSION : 1.0
// stored: InstanceOfName IEC_TIMER
"IEC_TIMER"
BEGIN
END_DATA_BLOCK

DATA_BLOCK "AI_3_5_Lolo_Timer"   // DB50
{ S7_Optimized_Access := 'TRUE' }
AUTHOR : Simatic
FAMILY : IEC
NAME : IEC_TMR
VERSION : 1.0
// stored: InstanceOfName IEC_TIMER
"IEC_TIMER"
BEGIN
END_DATA_BLOCK

DATA_BLOCK "AI_3_3_Lolo_Timer"   // DB51
{ S7_Optimized_Access := 'TRUE' }
AUTHOR : Simatic
FAMILY : IEC
NAME : IEC_TMR
VERSION : 1.0
// stored: InstanceOfName IEC_TIMER
"IEC_TIMER"
BEGIN
END_DATA_BLOCK

DATA_BLOCK "AI_3_7_Lolo_Timer"   // DB52
{ S7_Optimized_Access := 'TRUE' }
AUTHOR : Simatic
FAMILY : IEC
NAME : IEC_TMR
VERSION : 1.0
// stored: InstanceOfName IEC_TIMER
"IEC_TIMER"
BEGIN
END_DATA_BLOCK

DATA_BLOCK "AI_3_6_Lolo_Timer"   // DB53
{ S7_Optimized_Access := 'TRUE' }
AUTHOR : Simatic
FAMILY : IEC
NAME : IEC_TMR
VERSION : 1.0
// stored: InstanceOfName IEC_TIMER
"IEC_TIMER"
BEGIN
END_DATA_BLOCK

DATA_BLOCK "AI_2_1_Hihi_Timer"   // DB54
{ S7_Optimized_Access := 'TRUE' }
AUTHOR : Simatic
FAMILY : IEC
NAME : IEC_TMR
VERSION : 1.0
// stored: InstanceOfName IEC_TIMER
"IEC_TIMER"
BEGIN
END_DATA_BLOCK

DATA_BLOCK "AI_2_2_Hihi_Timer"   // DB55
{ S7_Optimized_Access := 'TRUE' }
AUTHOR : Simatic
FAMILY : IEC
NAME : IEC_TMR
VERSION : 1.0
// stored: InstanceOfName IEC_TIMER
"IEC_TIMER"
BEGIN
END_DATA_BLOCK

DATA_BLOCK "AI_3_2_Lolo_Timer"   // DB56
{ S7_Optimized_Access := 'TRUE' }
AUTHOR : Simatic
FAMILY : IEC
NAME : IEC_TMR
VERSION : 1.0
// stored: InstanceOfName IEC_TIMER
"IEC_TIMER"
BEGIN
END_DATA_BLOCK

DATA_BLOCK "AI_3_4_Lolo_Timer"   // DB57
{ S7_Optimized_Access := 'TRUE' }
AUTHOR : Simatic
FAMILY : IEC
NAME : IEC_TMR
VERSION : 1.0
// stored: InstanceOfName IEC_TIMER
"IEC_TIMER"
BEGIN
END_DATA_BLOCK

DATA_BLOCK "AI_3_3_Overflow_Timer"   // DB58
{ S7_Optimized_Access := 'TRUE' }
AUTHOR : Simatic
FAMILY : IEC
NAME : IEC_TMR
VERSION : 1.0
// stored: InstanceOfName IEC_TIMER
"IEC_TIMER"
BEGIN
END_DATA_BLOCK

DATA_BLOCK "AI_3_7_Overflow_Timer"   // DB59
{ S7_Optimized_Access := 'TRUE' }
AUTHOR : Simatic
FAMILY : IEC
NAME : IEC_TMR
VERSION : 1.0
// stored: InstanceOfName IEC_TIMER
"IEC_TIMER"
BEGIN
END_DATA_BLOCK

DATA_BLOCK "AI_3_6_Overflow_Timer"   // DB60
{ S7_Optimized_Access := 'TRUE' }
AUTHOR : Simatic
FAMILY : IEC
NAME : IEC_TMR
VERSION : 1.0
// stored: InstanceOfName IEC_TIMER
"IEC_TIMER"
BEGIN
END_DATA_BLOCK

DATA_BLOCK "AI_3_4_Overflow_Timer"   // DB61
{ S7_Optimized_Access := 'TRUE' }
AUTHOR : Simatic
FAMILY : IEC
NAME : IEC_TMR
VERSION : 1.0
// stored: InstanceOfName IEC_TIMER
"IEC_TIMER"
BEGIN
END_DATA_BLOCK

DATA_BLOCK "AI_3_2_Overflow_Timer"   // DB62
{ S7_Optimized_Access := 'TRUE' }
AUTHOR : Simatic
FAMILY : IEC
NAME : IEC_TMR
VERSION : 1.0
// stored: InstanceOfName IEC_TIMER
"IEC_TIMER"
BEGIN
END_DATA_BLOCK

DATA_BLOCK "AI_3_5_Overflow_Timer"   // DB63
{ S7_Optimized_Access := 'TRUE' }
AUTHOR : Simatic
FAMILY : IEC
NAME : IEC_TMR
VERSION : 1.0
// stored: InstanceOfName IEC_TIMER
"IEC_TIMER"
BEGIN
END_DATA_BLOCK

DATA_BLOCK "AI_2_3_Hihi_Timer"   // DB64
{ S7_Optimized_Access := 'TRUE' }
AUTHOR : Simatic
FAMILY : IEC
NAME : IEC_TMR
VERSION : 1.0
// stored: InstanceOfName IEC_TIMER
"IEC_TIMER"
BEGIN
END_DATA_BLOCK

DATA_BLOCK "AI_3_4_WB_Timer"   // DB65
{ S7_Optimized_Access := 'TRUE' }
AUTHOR : Simatic
FAMILY : IEC
NAME : IEC_TMR
VERSION : 1.0
// stored: InstanceOfName IEC_TIMER
"IEC_TIMER"
BEGIN
END_DATA_BLOCK

DATA_BLOCK "AI_3_5_WB_Timer"   // DB66
{ S7_Optimized_Access := 'TRUE' }
AUTHOR : Simatic
FAMILY : IEC
NAME : IEC_TMR
VERSION : 1.0
// stored: InstanceOfName IEC_TIMER
"IEC_TIMER"
BEGIN
END_DATA_BLOCK

DATA_BLOCK "AI_3_7_WB_Timer"   // DB67
{ S7_Optimized_Access := 'TRUE' }
AUTHOR : Simatic
FAMILY : IEC
NAME : IEC_TMR
VERSION : 1.0
// stored: InstanceOfName IEC_TIMER
"IEC_TIMER"
BEGIN
END_DATA_BLOCK

DATA_BLOCK "AI_3_2_WB_Timer"   // DB68
{ S7_Optimized_Access := 'TRUE' }
AUTHOR : Simatic
FAMILY : IEC
NAME : IEC_TMR
VERSION : 1.0
// stored: InstanceOfName IEC_TIMER
"IEC_TIMER"
BEGIN
END_DATA_BLOCK

DATA_BLOCK "AI_3_3_WB_Timer"   // DB69
{ S7_Optimized_Access := 'TRUE' }
AUTHOR : Simatic
FAMILY : IEC
NAME : IEC_TMR
VERSION : 1.0
// stored: InstanceOfName IEC_TIMER
"IEC_TIMER"
BEGIN
END_DATA_BLOCK

DATA_BLOCK "AI_3_6_WB_Timer"   // DB70
{ S7_Optimized_Access := 'TRUE' }
AUTHOR : Simatic
FAMILY : IEC
NAME : IEC_TMR
VERSION : 1.0
// stored: InstanceOfName IEC_TIMER
"IEC_TIMER"
BEGIN
END_DATA_BLOCK

DATA_BLOCK "AI_2_4_Hihi_Timer"   // DB71
{ S7_Optimized_Access := 'TRUE' }
AUTHOR : Simatic
FAMILY : IEC
NAME : IEC_TMR
VERSION : 1.0
// stored: InstanceOfName IEC_TIMER
"IEC_TIMER"
BEGIN
END_DATA_BLOCK

DATA_BLOCK "AI_2_5_Hihi_Timer"   // DB85
{ S7_Optimized_Access := 'TRUE' }
AUTHOR : Simatic
FAMILY : IEC
NAME : IEC_TMR
VERSION : 1.0
// stored: InstanceOfName IEC_TIMER
"IEC_TIMER"
BEGIN
END_DATA_BLOCK

DATA_BLOCK "AI_2_6_Hihi_Timer"   // DB86
{ S7_Optimized_Access := 'TRUE' }
AUTHOR : Simatic
FAMILY : IEC
NAME : IEC_TMR
VERSION : 1.0
// stored: InstanceOfName IEC_TIMER
"IEC_TIMER"
BEGIN
END_DATA_BLOCK

DATA_BLOCK "AI_2_7_Hihi_Timer"   // DB87
{ S7_Optimized_Access := 'TRUE' }
AUTHOR : Simatic
FAMILY : IEC
NAME : IEC_TMR
VERSION : 1.0
// stored: InstanceOfName IEC_TIMER
"IEC_TIMER"
BEGIN
END_DATA_BLOCK

DATA_BLOCK "AI_3_0_Hihi_Timer"   // DB88
{ S7_Optimized_Access := 'TRUE' }
AUTHOR : Simatic
FAMILY : IEC
NAME : IEC_TMR
VERSION : 1.0
// stored: InstanceOfName IEC_TIMER
"IEC_TIMER"
BEGIN
END_DATA_BLOCK

DATA_BLOCK "AI_3_1_Hihi_Timer"   // DB89
{ S7_Optimized_Access := 'TRUE' }
AUTHOR : Simatic
FAMILY : IEC
NAME : IEC_TMR
VERSION : 1.0
// stored: InstanceOfName IEC_TIMER
"IEC_TIMER"
BEGIN
END_DATA_BLOCK

DATA_BLOCK "AI_2_1_High_Timer"   // DB98
{ S7_Optimized_Access := 'TRUE' }
AUTHOR : Simatic
FAMILY : IEC
NAME : IEC_TMR
VERSION : 1.0
// stored: InstanceOfName IEC_TIMER
"IEC_TIMER"
BEGIN
END_DATA_BLOCK

DATA_BLOCK "AI_2_2_High_Timer"   // DB99
{ S7_Optimized_Access := 'TRUE' }
AUTHOR : Simatic
FAMILY : IEC
NAME : IEC_TMR
VERSION : 1.0
// stored: InstanceOfName IEC_TIMER
"IEC_TIMER"
BEGIN
END_DATA_BLOCK

DATA_BLOCK "AI_2_3_High_Timer"   // DB100
{ S7_Optimized_Access := 'TRUE' }
AUTHOR : Simatic
FAMILY : IEC
NAME : IEC_TMR
VERSION : 1.0
// stored: InstanceOfName IEC_TIMER
"IEC_TIMER"
BEGIN
END_DATA_BLOCK

DATA_BLOCK "AI_2_4_High_Timer"   // DB101
{ S7_Optimized_Access := 'TRUE' }
AUTHOR : Simatic
FAMILY : IEC
NAME : IEC_TMR
VERSION : 1.0
// stored: InstanceOfName IEC_TIMER
"IEC_TIMER"
BEGIN
END_DATA_BLOCK

DATA_BLOCK "AI_2_5_High_Timer"   // DB102
{ S7_Optimized_Access := 'TRUE' }
AUTHOR : Simatic
FAMILY : IEC
NAME : IEC_TMR
VERSION : 1.0
// stored: InstanceOfName IEC_TIMER
"IEC_TIMER"
BEGIN
END_DATA_BLOCK

DATA_BLOCK "AI_2_6_High_Timer"   // DB103
{ S7_Optimized_Access := 'TRUE' }
AUTHOR : Simatic
FAMILY : IEC
NAME : IEC_TMR
VERSION : 1.0
// stored: InstanceOfName IEC_TIMER
"IEC_TIMER"
BEGIN
END_DATA_BLOCK

DATA_BLOCK "AI_2_7_High_Timer"   // DB104
{ S7_Optimized_Access := 'TRUE' }
AUTHOR : Simatic
FAMILY : IEC
NAME : IEC_TMR
VERSION : 1.0
// stored: InstanceOfName IEC_TIMER
"IEC_TIMER"
BEGIN
END_DATA_BLOCK

DATA_BLOCK "AI_3_0_High_Timer"   // DB105
{ S7_Optimized_Access := 'TRUE' }
AUTHOR : Simatic
FAMILY : IEC
NAME : IEC_TMR
VERSION : 1.0
// stored: InstanceOfName IEC_TIMER
"IEC_TIMER"
BEGIN
END_DATA_BLOCK

DATA_BLOCK "AI_3_1_High_Timer"   // DB106
{ S7_Optimized_Access := 'TRUE' }
AUTHOR : Simatic
FAMILY : IEC
NAME : IEC_TMR
VERSION : 1.0
// stored: InstanceOfName IEC_TIMER
"IEC_TIMER"
BEGIN
END_DATA_BLOCK

DATA_BLOCK "AI_2_1_Low_Timer"   // DB115
{ S7_Optimized_Access := 'TRUE' }
AUTHOR : Simatic
FAMILY : IEC
NAME : IEC_TMR
VERSION : 1.0
// stored: InstanceOfName IEC_TIMER
"IEC_TIMER"
BEGIN
END_DATA_BLOCK

DATA_BLOCK "AI_2_2_Low_Timer"   // DB116
{ S7_Optimized_Access := 'TRUE' }
AUTHOR : Simatic
FAMILY : IEC
NAME : IEC_TMR
VERSION : 1.0
// stored: InstanceOfName IEC_TIMER
"IEC_TIMER"
BEGIN
END_DATA_BLOCK

DATA_BLOCK "AI_2_3_Low_Timer"   // DB117
{ S7_Optimized_Access := 'TRUE' }
AUTHOR : Simatic
FAMILY : IEC
NAME : IEC_TMR
VERSION : 1.0
// stored: InstanceOfName IEC_TIMER
"IEC_TIMER"
BEGIN
END_DATA_BLOCK

DATA_BLOCK "AI_2_4_Low_Timer"   // DB118
{ S7_Optimized_Access := 'TRUE' }
AUTHOR : Simatic
FAMILY : IEC
NAME : IEC_TMR
VERSION : 1.0
// stored: InstanceOfName IEC_TIMER
"IEC_TIMER"
BEGIN
END_DATA_BLOCK

DATA_BLOCK "AI_2_5_Low_Timer"   // DB122
{ S7_Optimized_Access := 'TRUE' }
AUTHOR : Simatic
FAMILY : IEC
NAME : IEC_TMR
VERSION : 1.0
// stored: InstanceOfName IEC_TIMER
"IEC_TIMER"
BEGIN
END_DATA_BLOCK

DATA_BLOCK "AI_2_6_Low_Timer"   // DB123
{ S7_Optimized_Access := 'TRUE' }
AUTHOR : Simatic
FAMILY : IEC
NAME : IEC_TMR
VERSION : 1.0
// stored: InstanceOfName IEC_TIMER
"IEC_TIMER"
BEGIN
END_DATA_BLOCK

DATA_BLOCK "AI_2_7_Low_Timer"   // DB124
{ S7_Optimized_Access := 'TRUE' }
AUTHOR : Simatic
FAMILY : IEC
NAME : IEC_TMR
VERSION : 1.0
// stored: InstanceOfName IEC_TIMER
"IEC_TIMER"
BEGIN
END_DATA_BLOCK

DATA_BLOCK "AI_3_0_Low_Timer"   // DB125
{ S7_Optimized_Access := 'TRUE' }
AUTHOR : Simatic
FAMILY : IEC
NAME : IEC_TMR
VERSION : 1.0
// stored: InstanceOfName IEC_TIMER
"IEC_TIMER"
BEGIN
END_DATA_BLOCK

DATA_BLOCK "AI_3_1_Low_Timer"   // DB126
{ S7_Optimized_Access := 'TRUE' }
AUTHOR : Simatic
FAMILY : IEC
NAME : IEC_TMR
VERSION : 1.0
// stored: InstanceOfName IEC_TIMER
"IEC_TIMER"
BEGIN
END_DATA_BLOCK

DATA_BLOCK "AI_2_1_Lolo_Timer"   // DB135
{ S7_Optimized_Access := 'TRUE' }
AUTHOR : Simatic
FAMILY : IEC
NAME : IEC_TMR
VERSION : 1.0
// stored: InstanceOfName IEC_TIMER
"IEC_TIMER"
BEGIN
END_DATA_BLOCK

DATA_BLOCK "AI_2_2_Lolo_Timer"   // DB136
{ S7_Optimized_Access := 'TRUE' }
AUTHOR : Simatic
FAMILY : IEC
NAME : IEC_TMR
VERSION : 1.0
// stored: InstanceOfName IEC_TIMER
"IEC_TIMER"
BEGIN
END_DATA_BLOCK

DATA_BLOCK "AI_2_3_Lolo_Timer"   // DB137
{ S7_Optimized_Access := 'TRUE' }
AUTHOR : Simatic
FAMILY : IEC
NAME : IEC_TMR
VERSION : 1.0
// stored: InstanceOfName IEC_TIMER
"IEC_TIMER"
BEGIN
END_DATA_BLOCK

DATA_BLOCK "AI_2_4_Lolo_Timer"   // DB138
{ S7_Optimized_Access := 'TRUE' }
AUTHOR : Simatic
FAMILY : IEC
NAME : IEC_TMR
VERSION : 1.0
// stored: InstanceOfName IEC_TIMER
"IEC_TIMER"
BEGIN
END_DATA_BLOCK

DATA_BLOCK "AI_2_5_Lolo_Timer"   // DB139
{ S7_Optimized_Access := 'TRUE' }
AUTHOR : Simatic
FAMILY : IEC
NAME : IEC_TMR
VERSION : 1.0
// stored: InstanceOfName IEC_TIMER
"IEC_TIMER"
BEGIN
END_DATA_BLOCK

DATA_BLOCK "AI_2_6_Lolo_Timer"   // DB140
{ S7_Optimized_Access := 'TRUE' }
AUTHOR : Simatic
FAMILY : IEC
NAME : IEC_TMR
VERSION : 1.0
// stored: InstanceOfName IEC_TIMER
"IEC_TIMER"
BEGIN
END_DATA_BLOCK

DATA_BLOCK "AI_2_7_Lolo_Timer"   // DB141
{ S7_Optimized_Access := 'TRUE' }
AUTHOR : Simatic
FAMILY : IEC
NAME : IEC_TMR
VERSION : 1.0
// stored: InstanceOfName IEC_TIMER
"IEC_TIMER"
BEGIN
END_DATA_BLOCK

DATA_BLOCK "AI_3_0_Lolo_Timer"   // DB142
{ S7_Optimized_Access := 'TRUE' }
AUTHOR : Simatic
FAMILY : IEC
NAME : IEC_TMR
VERSION : 1.0
// stored: InstanceOfName IEC_TIMER
"IEC_TIMER"
BEGIN
END_DATA_BLOCK

DATA_BLOCK "AI_3_1_Lolo_Timer"   // DB143
{ S7_Optimized_Access := 'TRUE' }
AUTHOR : Simatic
FAMILY : IEC
NAME : IEC_TMR
VERSION : 1.0
// stored: InstanceOfName IEC_TIMER
"IEC_TIMER"
BEGIN
END_DATA_BLOCK

DATA_BLOCK "AI_2_1_Overflow_Timer"   // DB152
{ S7_Optimized_Access := 'TRUE' }
AUTHOR : Simatic
FAMILY : IEC
NAME : IEC_TMR
VERSION : 1.0
// stored: InstanceOfName IEC_TIMER
"IEC_TIMER"
BEGIN
END_DATA_BLOCK

DATA_BLOCK "AI_2_2_Overflow_Timer"   // DB153
{ S7_Optimized_Access := 'TRUE' }
AUTHOR : Simatic
FAMILY : IEC
NAME : IEC_TMR
VERSION : 1.0
// stored: InstanceOfName IEC_TIMER
"IEC_TIMER"
BEGIN
END_DATA_BLOCK

DATA_BLOCK "AI_2_3_Overflow_Timer"   // DB154
{ S7_Optimized_Access := 'TRUE' }
AUTHOR : Simatic
FAMILY : IEC
NAME : IEC_TMR
VERSION : 1.0
// stored: InstanceOfName IEC_TIMER
"IEC_TIMER"
BEGIN
END_DATA_BLOCK

DATA_BLOCK "AI_2_4_Overflow_Timer"   // DB155
{ S7_Optimized_Access := 'TRUE' }
AUTHOR : Simatic
FAMILY : IEC
NAME : IEC_TMR
VERSION : 1.0
// stored: InstanceOfName IEC_TIMER
"IEC_TIMER"
BEGIN
END_DATA_BLOCK

DATA_BLOCK "AI_2_5_Overflow_Timer"   // DB156
{ S7_Optimized_Access := 'TRUE' }
AUTHOR : Simatic
FAMILY : IEC
NAME : IEC_TMR
VERSION : 1.0
// stored: InstanceOfName IEC_TIMER
"IEC_TIMER"
BEGIN
END_DATA_BLOCK

DATA_BLOCK "AI_2_6_Overflow_Timer"   // DB157
{ S7_Optimized_Access := 'TRUE' }
AUTHOR : Simatic
FAMILY : IEC
NAME : IEC_TMR
VERSION : 1.0
// stored: InstanceOfName IEC_TIMER
"IEC_TIMER"
BEGIN
END_DATA_BLOCK

DATA_BLOCK "AI_2_7_Overflow_Timer"   // DB158
{ S7_Optimized_Access := 'TRUE' }
AUTHOR : Simatic
FAMILY : IEC
NAME : IEC_TMR
VERSION : 1.0
// stored: InstanceOfName IEC_TIMER
"IEC_TIMER"
BEGIN
END_DATA_BLOCK

DATA_BLOCK "AI_3_0_Overflow_Timer"   // DB159
{ S7_Optimized_Access := 'TRUE' }
AUTHOR : Simatic
FAMILY : IEC
NAME : IEC_TMR
VERSION : 1.0
// stored: InstanceOfName IEC_TIMER
"IEC_TIMER"
BEGIN
END_DATA_BLOCK

DATA_BLOCK "AI_3_1_Overflow_Timer"   // DB160
{ S7_Optimized_Access := 'TRUE' }
AUTHOR : Simatic
FAMILY : IEC
NAME : IEC_TMR
VERSION : 1.0
// stored: InstanceOfName IEC_TIMER
"IEC_TIMER"
BEGIN
END_DATA_BLOCK

DATA_BLOCK "AI_2_1_WB_Timer"   // DB169
{ S7_Optimized_Access := 'TRUE' }
AUTHOR : Simatic
FAMILY : IEC
NAME : IEC_TMR
VERSION : 1.0
// stored: InstanceOfName IEC_TIMER
"IEC_TIMER"
BEGIN
END_DATA_BLOCK

DATA_BLOCK "AI_2_2_WB_Timer"   // DB170
{ S7_Optimized_Access := 'TRUE' }
AUTHOR : Simatic
FAMILY : IEC
NAME : IEC_TMR
VERSION : 1.0
// stored: InstanceOfName IEC_TIMER
"IEC_TIMER"
BEGIN
END_DATA_BLOCK

DATA_BLOCK "AI_2_3_WB_Timer"   // DB171
{ S7_Optimized_Access := 'TRUE' }
AUTHOR : Simatic
FAMILY : IEC
NAME : IEC_TMR
VERSION : 1.0
// stored: InstanceOfName IEC_TIMER
"IEC_TIMER"
BEGIN
END_DATA_BLOCK

DATA_BLOCK "AI_2_4_WB_Timer"   // DB172
{ S7_Optimized_Access := 'TRUE' }
AUTHOR : Simatic
FAMILY : IEC
NAME : IEC_TMR
VERSION : 1.0
// stored: InstanceOfName IEC_TIMER
"IEC_TIMER"
BEGIN
END_DATA_BLOCK

DATA_BLOCK "AI_2_5_WB_Timer"   // DB173
{ S7_Optimized_Access := 'TRUE' }
AUTHOR : Simatic
FAMILY : IEC
NAME : IEC_TMR
VERSION : 1.0
// stored: InstanceOfName IEC_TIMER
"IEC_TIMER"
BEGIN
END_DATA_BLOCK

DATA_BLOCK "AI_2_6_WB_Timer"   // DB174
{ S7_Optimized_Access := 'TRUE' }
AUTHOR : Simatic
FAMILY : IEC
NAME : IEC_TMR
VERSION : 1.0
// stored: InstanceOfName IEC_TIMER
"IEC_TIMER"
BEGIN
END_DATA_BLOCK

DATA_BLOCK "AI_2_7_WB_Timer"   // DB175
{ S7_Optimized_Access := 'TRUE' }
AUTHOR : Simatic
FAMILY : IEC
NAME : IEC_TMR
VERSION : 1.0
// stored: InstanceOfName IEC_TIMER
"IEC_TIMER"
BEGIN
END_DATA_BLOCK

DATA_BLOCK "AI_3_0_WB_Timer"   // DB176
{ S7_Optimized_Access := 'TRUE' }
AUTHOR : Simatic
FAMILY : IEC
NAME : IEC_TMR
VERSION : 1.0
// stored: InstanceOfName IEC_TIMER
"IEC_TIMER"
BEGIN
END_DATA_BLOCK

DATA_BLOCK "AI_3_1_WB_Timer"   // DB177
{ S7_Optimized_Access := 'TRUE' }
AUTHOR : Simatic
FAMILY : IEC
NAME : IEC_TMR
VERSION : 1.0
// stored: InstanceOfName IEC_TIMER
"IEC_TIMER"
BEGIN
END_DATA_BLOCK

DATA_BLOCK "DI_1_4_TON"   // DB186
{ S7_Optimized_Access := 'TRUE' }
AUTHOR : Simatic
FAMILY : IEC
NAME : IEC_TMR
VERSION : 1.0
// stored: InstanceOfName IEC_TIMER
"IEC_TIMER"
BEGIN
END_DATA_BLOCK

DATA_BLOCK "DI_1_3_TON"   // DB187
{ S7_Optimized_Access := 'TRUE' }
AUTHOR : Simatic
FAMILY : IEC
NAME : IEC_TMR
VERSION : 1.0
// stored: InstanceOfName IEC_TIMER
"IEC_TIMER"
BEGIN
END_DATA_BLOCK

DATA_BLOCK "DI_1_6_TON"   // DB188
{ S7_Optimized_Access := 'TRUE' }
AUTHOR : Simatic
FAMILY : IEC
NAME : IEC_TMR
VERSION : 1.0
// stored: InstanceOfName IEC_TIMER
"IEC_TIMER"
BEGIN
END_DATA_BLOCK

DATA_BLOCK "DI_1_5_TON"   // DB189
{ S7_Optimized_Access := 'TRUE' }
AUTHOR : Simatic
FAMILY : IEC
NAME : IEC_TMR
VERSION : 1.0
// stored: InstanceOfName IEC_TIMER
"IEC_TIMER"
BEGIN
END_DATA_BLOCK

DATA_BLOCK "DI_1_7_TON"   // DB190
{ S7_Optimized_Access := 'TRUE' }
AUTHOR : Simatic
FAMILY : IEC
NAME : IEC_TMR
VERSION : 1.0
// stored: InstanceOfName IEC_TIMER
"IEC_TIMER"
BEGIN
END_DATA_BLOCK

DATA_BLOCK "DI_1_9_TON"   // DB191
{ S7_Optimized_Access := 'TRUE' }
AUTHOR : Simatic
FAMILY : IEC
NAME : IEC_TMR
VERSION : 1.0
// stored: InstanceOfName IEC_TIMER
"IEC_TIMER"
BEGIN
END_DATA_BLOCK

DATA_BLOCK "DI_1_8_TON"   // DB192
{ S7_Optimized_Access := 'TRUE' }
AUTHOR : Simatic
FAMILY : IEC
NAME : IEC_TMR
VERSION : 1.0
// stored: InstanceOfName IEC_TIMER
"IEC_TIMER"
BEGIN
END_DATA_BLOCK

DATA_BLOCK "DI_1_11_TON"   // DB193
{ S7_Optimized_Access := 'TRUE' }
AUTHOR : Simatic
FAMILY : IEC
NAME : IEC_TMR
VERSION : 1.0
// stored: InstanceOfName IEC_TIMER
"IEC_TIMER"
BEGIN
END_DATA_BLOCK

DATA_BLOCK "DI_1_8_TOF"   // DB196
{ S7_Optimized_Access := 'TRUE' }
AUTHOR : Simatic
FAMILY : IEC
NAME : IEC_TMR
VERSION : 1.0
// stored: InstanceOfName IEC_TIMER
"IEC_TIMER"
BEGIN
END_DATA_BLOCK

DATA_BLOCK "DO_1_0_TOF"   // DB199
{ S7_Optimized_Access := 'TRUE' }
AUTHOR : Simatic
FAMILY : IEC
NAME : IEC_TMR
VERSION : 1.0
// stored: InstanceOfName IEC_TIMER
"IEC_TIMER"
BEGIN
END_DATA_BLOCK

DATA_BLOCK "DO_1_8_TON"   // DB200
{ S7_Optimized_Access := 'TRUE' }
AUTHOR : Simatic
FAMILY : IEC
NAME : IEC_TMR
VERSION : 1.0
// stored: InstanceOfName IEC_TIMER
"IEC_TIMER"
BEGIN
END_DATA_BLOCK

DATA_BLOCK "DO_1_1_TOF"   // DB202
{ S7_Optimized_Access := 'TRUE' }
AUTHOR : Simatic
FAMILY : IEC
NAME : IEC_TMR
VERSION : 1.0
// stored: InstanceOfName IEC_TIMER
"IEC_TIMER"
BEGIN
END_DATA_BLOCK

DATA_BLOCK "DO_1_8_TOF"   // DB203
{ S7_Optimized_Access := 'TRUE' }
AUTHOR : Simatic
FAMILY : IEC
NAME : IEC_TMR
VERSION : 1.0
// stored: InstanceOfName IEC_TIMER
"IEC_TIMER"
BEGIN
END_DATA_BLOCK

DATA_BLOCK "DI_1_10_TON"   // DB208
{ S7_Optimized_Access := 'TRUE' }
AUTHOR : Simatic
FAMILY : IEC
NAME : IEC_TMR
VERSION : 1.0
// stored: InstanceOfName IEC_TIMER
"IEC_TIMER"
BEGIN
END_DATA_BLOCK

DATA_BLOCK "DI_1_7_TOF"   // DB211
{ S7_Optimized_Access := 'TRUE' }
AUTHOR : Simatic
FAMILY : IEC
NAME : IEC_TMR
VERSION : 1.0
// stored: InstanceOfName IEC_TIMER
"IEC_TIMER"
BEGIN
END_DATA_BLOCK

DATA_BLOCK "DO_1_0_TON"   // DB214
{ S7_Optimized_Access := 'TRUE' }
AUTHOR : Simatic
FAMILY : IEC
NAME : IEC_TMR
VERSION : 1.0
// stored: InstanceOfName IEC_TIMER
"IEC_TIMER"
BEGIN
END_DATA_BLOCK

DATA_BLOCK "DO_1_7_TON"   // DB215
{ S7_Optimized_Access := 'TRUE' }
AUTHOR : Simatic
FAMILY : IEC
NAME : IEC_TMR
VERSION : 1.0
// stored: InstanceOfName IEC_TIMER
"IEC_TIMER"
BEGIN
END_DATA_BLOCK

DATA_BLOCK "DO_1_7_TOF"   // DB218
{ S7_Optimized_Access := 'TRUE' }
AUTHOR : Simatic
FAMILY : IEC
NAME : IEC_TMR
VERSION : 1.0
// stored: InstanceOfName IEC_TIMER
"IEC_TIMER"
BEGIN
END_DATA_BLOCK

DATA_BLOCK "DI_1_13_TON"   // DB223
{ S7_Optimized_Access := 'TRUE' }
AUTHOR : Simatic
FAMILY : IEC
NAME : IEC_TMR
VERSION : 1.0
// stored: InstanceOfName IEC_TIMER
"IEC_TIMER"
BEGIN
END_DATA_BLOCK

DATA_BLOCK "DI_1_3_TOF"   // DB225
{ S7_Optimized_Access := 'TRUE' }
AUTHOR : Simatic
FAMILY : IEC
NAME : IEC_TMR
VERSION : 1.0
// stored: InstanceOfName IEC_TIMER
"IEC_TIMER"
BEGIN
END_DATA_BLOCK

DATA_BLOCK "DI_1_10_TOF"   // DB226
{ S7_Optimized_Access := 'TRUE' }
AUTHOR : Simatic
FAMILY : IEC
NAME : IEC_TMR
VERSION : 1.0
// stored: InstanceOfName IEC_TIMER
"IEC_TIMER"
BEGIN
END_DATA_BLOCK

DATA_BLOCK "DO_1_3_TON"   // DB229
{ S7_Optimized_Access := 'TRUE' }
AUTHOR : Simatic
FAMILY : IEC
NAME : IEC_TMR
VERSION : 1.0
// stored: InstanceOfName IEC_TIMER
"IEC_TIMER"
BEGIN
END_DATA_BLOCK

DATA_BLOCK "DO_2_0_TON"   // DB230
{ S7_Optimized_Access := 'TRUE' }
AUTHOR : Simatic
FAMILY : IEC
NAME : IEC_TMR
VERSION : 1.0
// stored: InstanceOfName IEC_TIMER
"IEC_TIMER"
BEGIN
END_DATA_BLOCK

DATA_BLOCK "DO_1_3_TOF"   // DB232
{ S7_Optimized_Access := 'TRUE' }
AUTHOR : Simatic
FAMILY : IEC
NAME : IEC_TMR
VERSION : 1.0
// stored: InstanceOfName IEC_TIMER
"IEC_TIMER"
BEGIN
END_DATA_BLOCK

DATA_BLOCK "DO_1_1_TON"   // DB233
{ S7_Optimized_Access := 'TRUE' }
AUTHOR : Simatic
FAMILY : IEC
NAME : IEC_TMR
VERSION : 1.0
// stored: InstanceOfName IEC_TIMER
"IEC_TIMER"
BEGIN
END_DATA_BLOCK

DATA_BLOCK "DI_1_12_TON"   // DB238
{ S7_Optimized_Access := 'TRUE' }
AUTHOR : Simatic
FAMILY : IEC
NAME : IEC_TMR
VERSION : 1.0
// stored: InstanceOfName IEC_TIMER
"IEC_TIMER"
BEGIN
END_DATA_BLOCK

DATA_BLOCK "DI_1_9_TOF"   // DB241
{ S7_Optimized_Access := 'TRUE' }
AUTHOR : Simatic
FAMILY : IEC
NAME : IEC_TMR
VERSION : 1.0
// stored: InstanceOfName IEC_TIMER
"IEC_TIMER"
BEGIN
END_DATA_BLOCK

